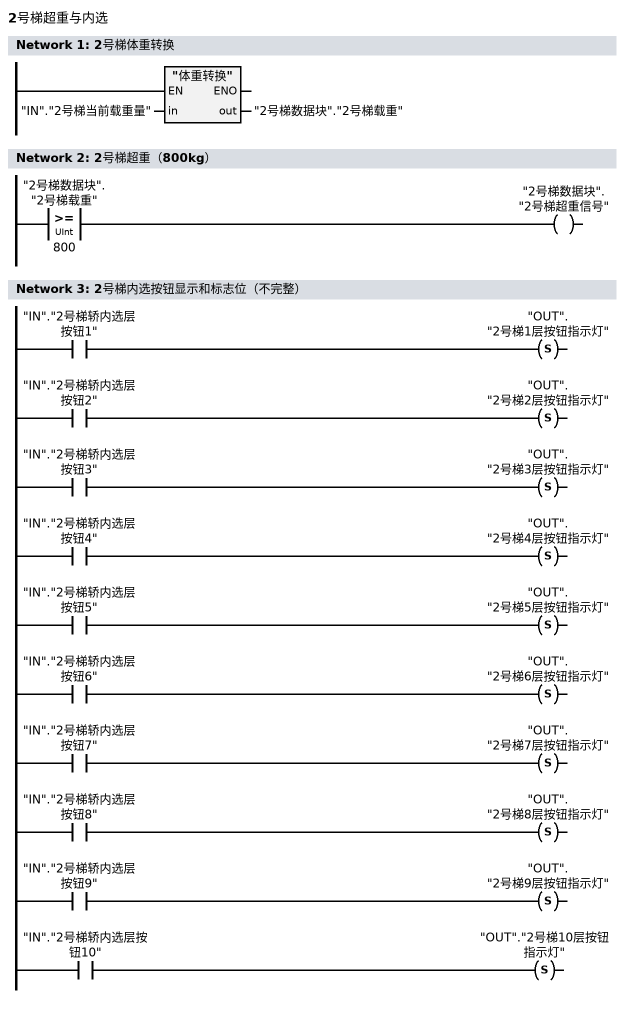
   RUNG wire#powerrail
      "体重转换"(in := "IN"."2号梯当前载重量", out => "2号梯数据块"."2号梯载重")
   END_RUNG
   // the same network as SCL:
   "体重转换"(in := "IN"."2号梯当前载重量", out => "2号梯数据块"."2号梯载重");
END_REGION

REGION Network 2: 2号梯超重（800kg）
   RUNG wire#powerrail
      { S7_Templates := "SrcType := UInt" } GE_Contact(in1 := "2号梯数据块"."2号梯载重", in2 := 800)
      Coil( "2号梯数据块"."2号梯超重信号" )
   END_RUNG
   // the same network as SCL:
   "2号梯数据块"."2号梯超重信号" := "2号梯数据块"."2号梯载重" >= 800;
END_REGION

REGION Network 3: 2号梯内选按钮显示和标志位（不完整）
   RUNG wire#powerrail
      Contact( "IN"."2号梯轿内选层按钮1" )
      S_Coil( "OUT"."2号梯1层按钮指示灯" )
   END_RUNG
   RUNG wire#powerrail
      Contact( "IN"."2号梯轿内选层按钮2" )
      S_Coil( "OUT"."2号梯2层按钮指示灯" )
   END_RUNG
   RUNG wire#powerrail
      Contact( "IN"."2号梯轿内选层按钮3" )
      S_Coil( "OUT"."2号梯3层按钮指示灯" )
   END_RUNG
   RUNG wire#powerrail
      Contact( "IN"."2号梯轿内选层按钮4" )
      S_Coil( "OUT"."2号梯4层按钮指示灯" )
   END_RUNG
   RUNG wire#powerrail
      Contact( "IN"."2号梯轿内选层按钮5" )
      S_Coil( "OUT"."2号梯5层按钮指示灯" )
   END_RUNG
   RUNG wire#powerrail
      Contact( "IN"."2号梯轿内选层按钮6" )
      S_Coil( "OUT"."2号梯6层按钮指示灯" )
   END_RUNG
   RUNG wire#powerrail
      Contact( "IN"."2号梯轿内选层按钮7" )
      S_Coil( "OUT"."2号梯7层按钮指示灯" )
   END_RUNG
   RUNG wire#powerrail
      Contact( "IN"."2号梯轿内选层按钮8" )
      S_Coil( "OUT"."2号梯8层按钮指示灯" )
   END_RUNG
   RUNG wire#powerrail
      Contact( "IN"."2号梯轿内选层按钮9" )
      S_Coil( "OUT"."2号梯9层按钮指示灯" )
   END_RUNG
   RUNG wire#powerrail
      Contact( "IN"."2号梯轿内选层按钮10" )
      S_Coil( "OUT"."2号梯10层按钮指示灯" )
   END_RUNG
   // the same network as SCL:
   IF "IN"."2号梯轿内选层按钮1" THEN "OUT"."2号梯1层按钮指示灯" := TRUE; END_IF;
   IF "IN"."2号梯轿内选层按钮2" THEN "OUT"."2号梯2层按钮指示灯" := TRUE; END_IF;
   IF "IN"."2号梯轿内选层按钮3" THEN "OUT"."2号梯3层按钮指示灯" := TRUE; END_IF;
   IF "IN"."2号梯轿内选层按钮4" THEN "OUT"."2号梯4层按钮指示灯" := TRUE; END_IF;
   IF "IN"."2号梯轿内选层按钮5" THEN "OUT"."2号梯5层按钮指示灯" := TRUE; END_IF;
   IF "IN"."2号梯轿内选层按钮6" THEN "OUT"."2号梯6层按钮指示灯" := TRUE; END_IF;
   IF "IN"."2号梯轿内选层按钮7" THEN "OUT"."2号梯7层按钮指示灯" := TRUE; END_IF;
   IF "IN"."2号梯轿内选层按钮8" THEN "OUT"."2号梯8层按钮指示灯" := TRUE; END_IF;
   IF "IN"."2号梯轿内选层按钮9" THEN "OUT"."2号梯9层按钮指示灯" := TRUE; END_IF;
   IF "IN"."2号梯轿内选层按钮10" THEN "OUT"."2号梯10层按钮指示灯" := TRUE; END_IF;
END_REGION
END_FUNCTION

FUNCTION "2号梯开关门控制" : Void   // FC27, LAD
{ S7_Optimized_Access := 'TRUE' }
VERSION : 0.1
BEGIN
END_FUNCTION

FUNCTION "2号梯楼层计数" : Void   // FC33, LAD
{ S7_Optimized_Access := 'TRUE' }
VERSION : 0.1
BEGIN
END_FUNCTION

FUNCTION "2号梯检修" : Void   // FC44, LAD
{ S7_Optimized_Access := 'TRUE' }
VERSION : 0.1
BEGIN
END_FUNCTION

FUNCTION "2号梯目标楼层与方向判断" : Void   // FC45, LAD
{ S7_Optimized_Access := 'TRUE' }
VERSION : 0.1
BEGIN
END_FUNCTION

FUNCTION "2号梯字节消除与记录" : Void   // FC46, LAD
{ S7_Optimized_Access := 'TRUE' }
VERSION : 0.1
BEGIN
END_FUNCTION

FUNCTION "2号梯启停控制" : Void   // FC59, LAD
{ S7_Optimized_Access := 'TRUE' }
VERSION : 0.1
BEGIN
END_FUNCTION

// folder: 3号梯

FUNCTION "3号梯初始化" : Void   // FC4, LAD
{ S7_Optimized_Access := 'TRUE' }
VERSION : 0.1
   VAR_INPUT
      初始化方向 : Bool;
      初始化楼层 : Byte;
   END_VAR
   VAR_TEMP   // added for the SCL form of the ladder/FBD networks
      _w1 : Bool;
      _w2 : Bool;
      _w3 : Bool;
      _w4 : Bool;
   END_VAR
BEGIN

REGION Network 1: 3号梯传参（方向+初始化楼层）
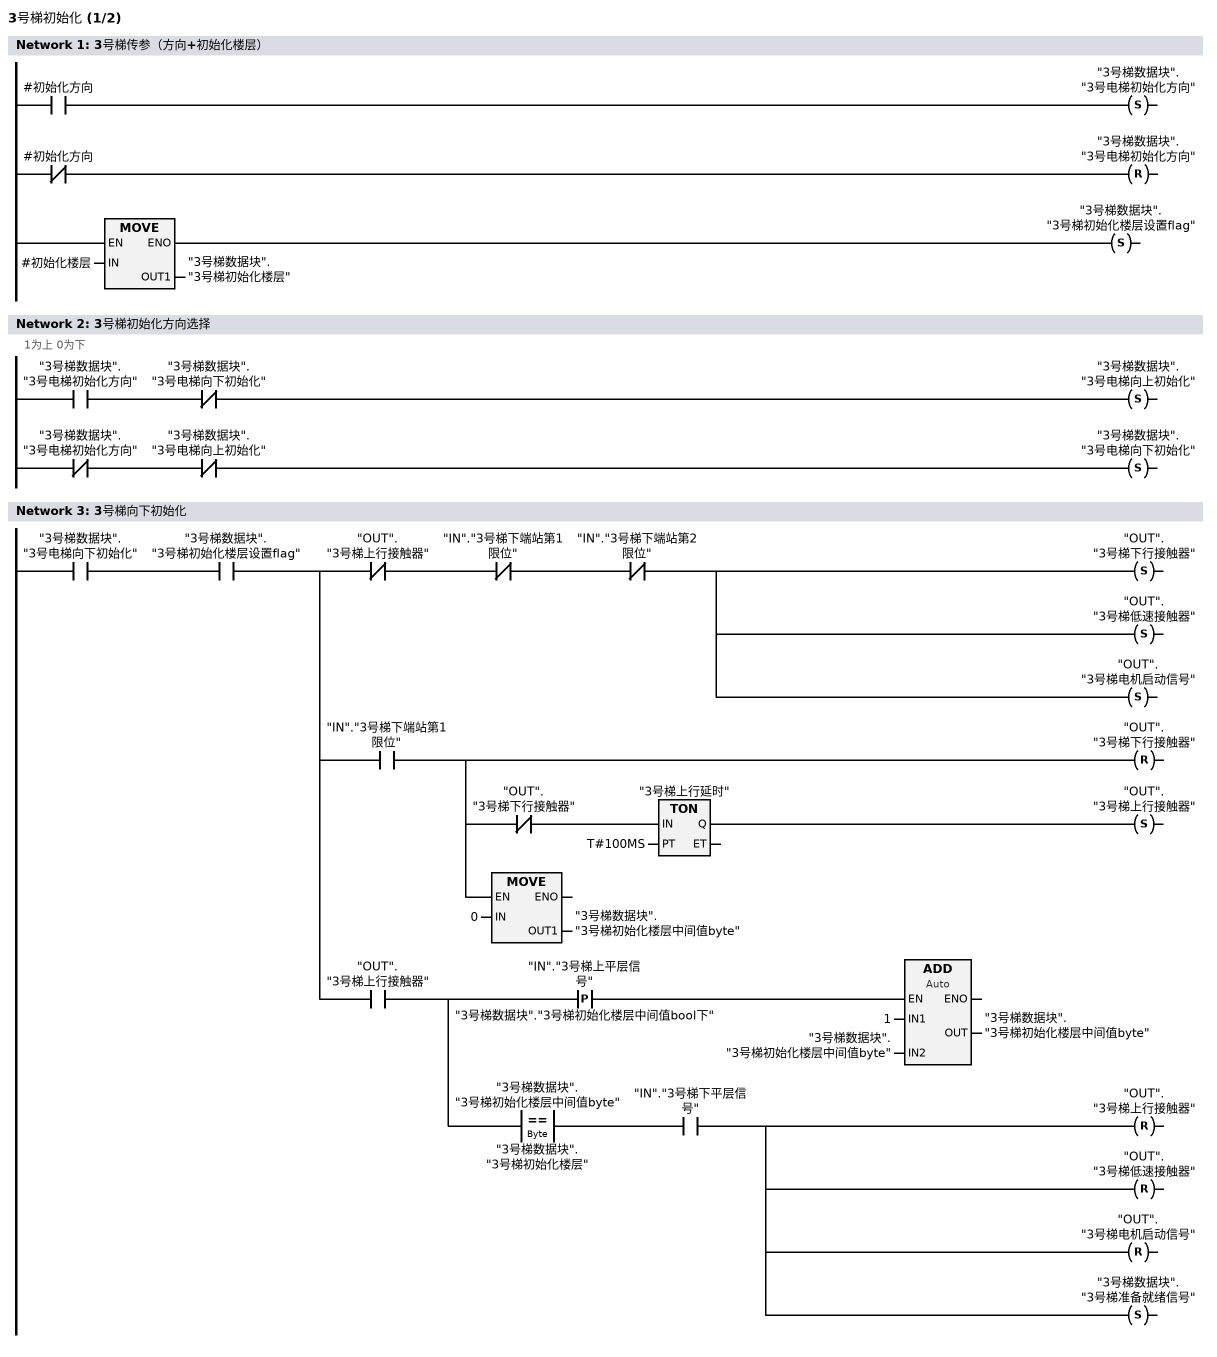
   RUNG wire#powerrail
      Contact( #初始化方向 )
      S_Coil( "3号梯数据块"."3号电梯初始化方向" )
   END_RUNG
   RUNG wire#powerrail
      I_Contact( #初始化方向 )
      R_Coil( "3号梯数据块"."3号电梯初始化方向" )
   END_RUNG
   RUNG wire#powerrail
      Move(in := #初始化楼层, out1 => "3号梯数据块"."3号梯初始化楼层")
      S_Coil( "3号梯数据块"."3号梯初始化楼层设置flag" )
   END_RUNG
   // the same network as SCL:
   IF #初始化方向 THEN "3号梯数据块"."3号电梯初始化方向" := TRUE; END_IF;
   IF NOT #初始化方向 THEN "3号梯数据块"."3号电梯初始化方向" := FALSE; END_IF;
   "3号梯数据块"."3号梯初始化楼层" := #初始化楼层;
   "3号梯数据块"."3号梯初始化楼层设置flag" := TRUE;
END_REGION

REGION Network 2: 3号梯初始化方向选择
   // 1为上 0为下
   RUNG wire#powerrail
      Contact( "3号梯数据块"."3号电梯初始化方向" )
      I_Contact( "3号梯数据块"."3号电梯向下初始化" )
      S_Coil( "3号梯数据块"."3号电梯向上初始化" )
   END_RUNG
   RUNG wire#powerrail
      I_Contact( "3号梯数据块"."3号电梯初始化方向" )
      I_Contact( "3号梯数据块"."3号电梯向上初始化" )
      S_Coil( "3号梯数据块"."3号电梯向下初始化" )
   END_RUNG
   // the same network as SCL:
   IF "3号梯数据块"."3号电梯初始化方向" AND NOT "3号梯数据块"."3号电梯向下初始化" THEN "3号梯数据块"."3号电梯向上初始化" := TRUE; END_IF;
   IF NOT "3号梯数据块"."3号电梯初始化方向" AND NOT "3号梯数据块"."3号电梯向上初始化" THEN "3号梯数据块"."3号电梯向下初始化" := TRUE; END_IF;
END_REGION

REGION Network 3: 3号梯向下初始化
   #_w1 := "3号梯数据块"."3号电梯向下初始化" AND "3号梯数据块"."3号梯初始化楼层设置flag";
   IF #_w1 AND NOT "OUT"."3号梯上行接触器" AND NOT "IN"."3号梯下端站第1限位" AND NOT "IN"."3号梯下端站第2限位" THEN
       "OUT"."3号梯下行接触器" := TRUE;
       "OUT"."3号梯低速接触器" := TRUE;
       "OUT"."3号梯电机启动信号" := TRUE;
   END_IF;
   #_w2 := #_w1 AND "IN"."3号梯下端站第1限位";
   IF #_w2 THEN "OUT"."3号梯下行接触器" := FALSE; END_IF;
   "3号梯上行延时".TON(IN := #_w2 AND NOT "OUT"."3号梯下行接触器", PT := T#100MS);
   IF "3号梯上行延时".Q THEN "OUT"."3号梯上行接触器" := TRUE; END_IF;
   IF #_w2 THEN "3号梯数据块"."3号梯初始化楼层中间值byte" := 0; END_IF;
   #_w3 := #_w1 AND "OUT"."3号梯上行接触器";
   #_w4 := #_w3 AND "IN"."3号梯上平层信号" AND NOT "3号梯数据块"."3号梯初始化楼层中间值bool下";   // rising edge of "IN"."3号梯上平层信号"
   "3号梯数据块"."3号梯初始化楼层中间值bool下" := "IN"."3号梯上平层信号";
   IF #_w4 THEN "3号梯数据块"."3号梯初始化楼层中间值byte" := 1 + "3号梯数据块"."3号梯初始化楼层中间值byte"; END_IF;
   IF #_w3 AND ("3号梯数据块"."3号梯初始化楼层中间值byte" = "3号梯数据块"."3号梯初始化楼层") AND "IN"."3号梯下平层信号" THEN
       "OUT"."3号梯上行接触器" := FALSE;
       "OUT"."3号梯低速接触器" := FALSE;
       "OUT"."3号梯电机启动信号" := FALSE;
       "3号梯数据块"."3号梯准备就绪信号" := TRUE;
   END_IF;
END_REGION

REGION Network 4: 3号梯向上初始化
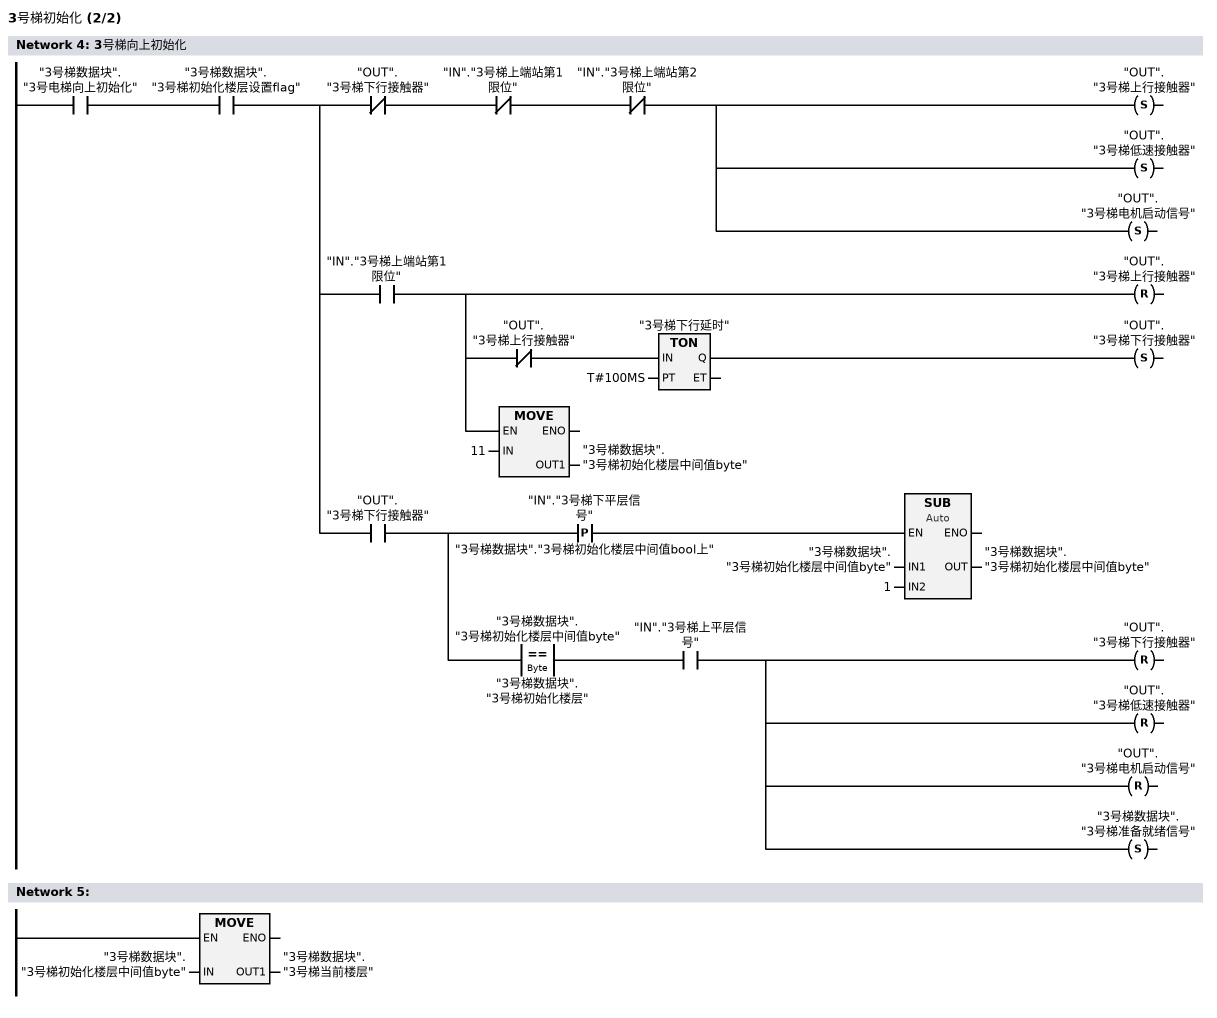
   #_w1 := "3号梯数据块"."3号电梯向上初始化" AND "3号梯数据块"."3号梯初始化楼层设置flag";
   IF #_w1 AND NOT "OUT"."3号梯下行接触器" AND NOT "IN"."3号梯上端站第1限位" AND NOT "IN"."3号梯上端站第2限位" THEN
       "OUT"."3号梯上行接触器" := TRUE;
       "OUT"."3号梯低速接触器" := TRUE;
       "OUT"."3号梯电机启动信号" := TRUE;
   END_IF;
   #_w2 := #_w1 AND "IN"."3号梯上端站第1限位";
   IF #_w2 THEN "OUT"."3号梯上行接触器" := FALSE; END_IF;
   "3号梯下行延时".TON(IN := #_w2 AND NOT "OUT"."3号梯上行接触器", PT := T#100MS);
   IF "3号梯下行延时".Q THEN "OUT"."3号梯下行接触器" := TRUE; END_IF;
   IF #_w2 THEN "3号梯数据块"."3号梯初始化楼层中间值byte" := 11; END_IF;
   #_w3 := #_w1 AND "OUT"."3号梯下行接触器";
   #_w4 := #_w3 AND "IN"."3号梯下平层信号" AND NOT "3号梯数据块"."3号梯初始化楼层中间值bool上";   // rising edge of "IN"."3号梯下平层信号"
   "3号梯数据块"."3号梯初始化楼层中间值bool上" := "IN"."3号梯下平层信号";
   IF #_w4 THEN "3号梯数据块"."3号梯初始化楼层中间值byte" := "3号梯数据块"."3号梯初始化楼层中间值byte" - 1; END_IF;
   IF #_w3 AND ("3号梯数据块"."3号梯初始化楼层中间值byte" = "3号梯数据块"."3号梯初始化楼层") AND "IN"."3号梯上平层信号" THEN
       "OUT"."3号梯下行接触器" := FALSE;
       "OUT"."3号梯低速接触器" := FALSE;
       "OUT"."3号梯电机启动信号" := FALSE;
       "3号梯数据块"."3号梯准备就绪信号" := TRUE;
   END_IF;
END_REGION

REGION Network 5
   RUNG wire#powerrail
      Move(in := "3号梯数据块"."3号梯初始化楼层中间值byte", out1 => "3号梯数据块"."3号梯当前楼层")
   END_RUNG
   // the same network as SCL:
   "3号梯数据块"."3号梯当前楼层" := "3号梯数据块"."3号梯初始化楼层中间值byte";
END_REGION
END_FUNCTION

FUNCTION "3号梯主函数" : Void   // FC10, LAD
{ S7_Optimized_Access := 'TRUE' }
VERSION : 0.1
BEGIN

REGION Network 1
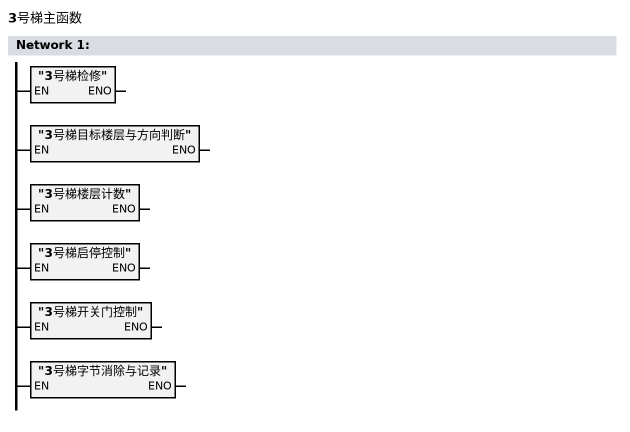
   RUNG wire#powerrail
      "3号梯检修"()
   END_RUNG
   RUNG wire#powerrail
      "3号梯目标楼层与方向判断"()
   END_RUNG
   RUNG wire#powerrail
      "3号梯楼层计数"()
   END_RUNG
   RUNG wire#powerrail
      "3号梯启停控制"()
   END_RUNG
   RUNG wire#powerrail
      "3号梯开关门控制"()
   END_RUNG
   RUNG wire#powerrail
      "3号梯字节消除与记录"()
   END_RUNG
   // the same network as SCL:
   "3号梯检修"();
   "3号梯目标楼层与方向判断"();
   "3号梯楼层计数"();
   "3号梯启停控制"();
   "3号梯开关门控制"();
   "3号梯字节消除与记录"();
END_REGION
END_FUNCTION

FUNCTION "3号梯运行监控模块" : Void   // FC16, LAD
{ S7_Optimized_Access := 'TRUE' }
VERSION : 0.1
BEGIN

REGION Network 1: 3号梯获取当前楼层设置标志位
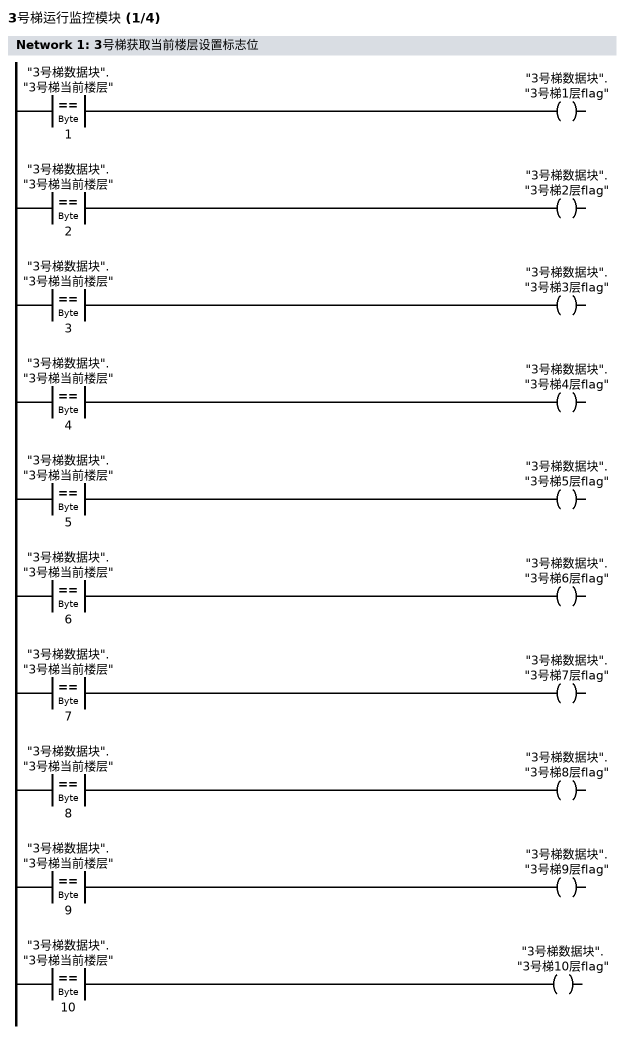
   RUNG wire#powerrail
      { S7_Templates := "SrcType := Byte" } EQ_Contact(in1 := "3号梯数据块"."3号梯当前楼层", in2 := 1)
      Coil( "3号梯数据块"."3号梯1层flag" )
   END_RUNG
   RUNG wire#powerrail
      { S7_Templates := "SrcType := Byte" } EQ_Contact(in1 := "3号梯数据块"."3号梯当前楼层", in2 := 2)
      Coil( "3号梯数据块"."3号梯2层flag" )
   END_RUNG
   RUNG wire#powerrail
      { S7_Templates := "SrcType := Byte" } EQ_Contact(in1 := "3号梯数据块"."3号梯当前楼层", in2 := 3)
      Coil( "3号梯数据块"."3号梯3层flag" )
   END_RUNG
   RUNG wire#powerrail
      { S7_Templates := "SrcType := Byte" } EQ_Contact(in1 := "3号梯数据块"."3号梯当前楼层", in2 := 4)
      Coil( "3号梯数据块"."3号梯4层flag" )
   END_RUNG
   RUNG wire#powerrail
      { S7_Templates := "SrcType := Byte" } EQ_Contact(in1 := "3号梯数据块"."3号梯当前楼层", in2 := 5)
      Coil( "3号梯数据块"."3号梯5层flag" )
   END_RUNG
   RUNG wire#powerrail
      { S7_Templates := "SrcType := Byte" } EQ_Contact(in1 := "3号梯数据块"."3号梯当前楼层", in2 := 6)
      Coil( "3号梯数据块"."3号梯6层flag" )
   END_RUNG
   RUNG wire#powerrail
      { S7_Templates := "SrcType := Byte" } EQ_Contact(in1 := "3号梯数据块"."3号梯当前楼层", in2 := 7)
      Coil( "3号梯数据块"."3号梯7层flag" )
   END_RUNG
   RUNG wire#powerrail
      { S7_Templates := "SrcType := Byte" } EQ_Contact(in1 := "3号梯数据块"."3号梯当前楼层", in2 := 8)
      Coil( "3号梯数据块"."3号梯8层flag" )
   END_RUNG
   RUNG wire#powerrail
      { S7_Templates := "SrcType := Byte" } EQ_Contact(in1 := "3号梯数据块"."3号梯当前楼层", in2 := 9)
      Coil( "3号梯数据块"."3号梯9层flag" )
   END_RUNG
   RUNG wire#powerrail
      { S7_Templates := "SrcType := Byte" } EQ_Contact(in1 := "3号梯数据块"."3号梯当前楼层", in2 := 10)
      Coil( "3号梯数据块"."3号梯10层flag" )
   END_RUNG
   // the same network as SCL:
   "3号梯数据块"."3号梯1层flag" := "3号梯数据块"."3号梯当前楼层" = 1;
   "3号梯数据块"."3号梯2层flag" := "3号梯数据块"."3号梯当前楼层" = 2;
   "3号梯数据块"."3号梯3层flag" := "3号梯数据块"."3号梯当前楼层" = 3;
   "3号梯数据块"."3号梯4层flag" := "3号梯数据块"."3号梯当前楼层" = 4;
   "3号梯数据块"."3号梯5层flag" := "3号梯数据块"."3号梯当前楼层" = 5;
   "3号梯数据块"."3号梯6层flag" := "3号梯数据块"."3号梯当前楼层" = 6;
   "3号梯数据块"."3号梯7层flag" := "3号梯数据块"."3号梯当前楼层" = 7;
   "3号梯数据块"."3号梯8层flag" := "3号梯数据块"."3号梯当前楼层" = 8;
   "3号梯数据块"."3号梯9层flag" := "3号梯数据块"."3号梯当前楼层" = 9;
   "3号梯数据块"."3号梯10层flag" := "3号梯数据块"."3号梯当前楼层" = 10;
END_REGION

REGION Network 2: 3号梯楼层led_a显示
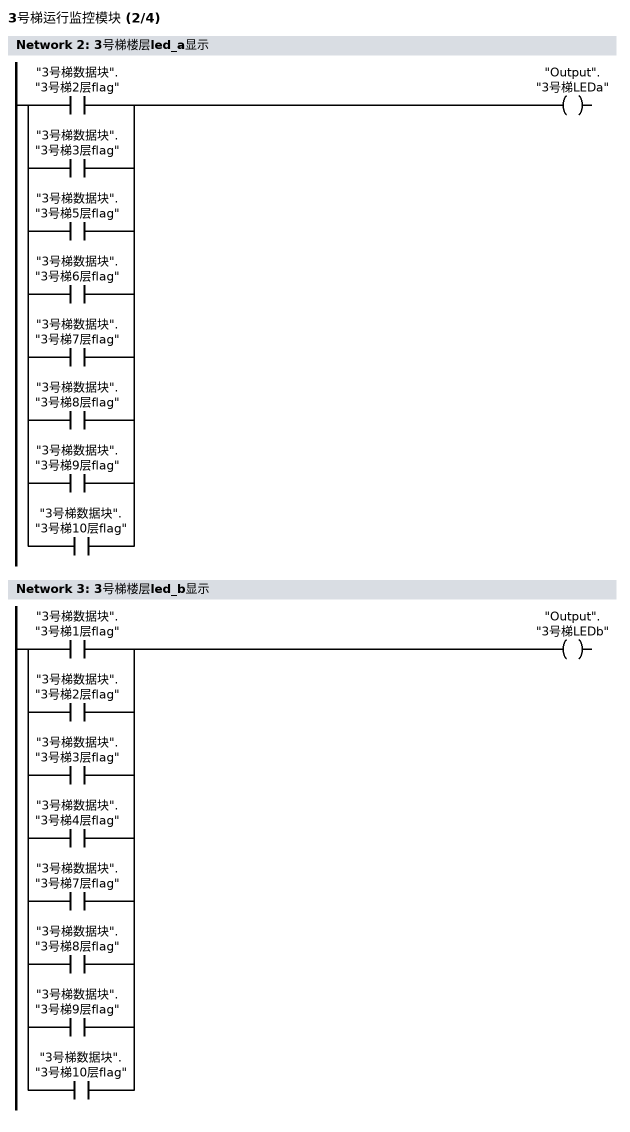
   RUNG wire#powerrail
      Contact( "3号梯数据块"."3号梯2层flag" )
      wire#w1
      Coil( "Output"."3号梯LEDa" )
   END_RUNG
   RUNG wire#powerrail
      Contact( "3号梯数据块"."3号梯3层flag" )
   END_RUNG wire#w1
   RUNG wire#powerrail
      Contact( "3号梯数据块"."3号梯5层flag" )
   END_RUNG wire#w1
   RUNG wire#powerrail
      Contact( "3号梯数据块"."3号梯6层flag" )
   END_RUNG wire#w1
   RUNG wire#powerrail
      Contact( "3号梯数据块"."3号梯7层flag" )
   END_RUNG wire#w1
   RUNG wire#powerrail
      Contact( "3号梯数据块"."3号梯8层flag" )
   END_RUNG wire#w1
   RUNG wire#powerrail
      Contact( "3号梯数据块"."3号梯9层flag" )
   END_RUNG wire#w1
   RUNG wire#powerrail
      Contact( "3号梯数据块"."3号梯10层flag" )
   END_RUNG wire#w1
   // the same network as SCL:
   "Output"."3号梯LEDa" := "3号梯数据块"."3号梯2层flag" OR "3号梯数据块"."3号梯3层flag" OR "3号梯数据块"."3号梯5层flag" OR "3号梯数据块"."3号梯6层flag" OR "3号梯数据块"."3号梯7层flag" OR "3号梯数据块"."3号梯8层flag" OR "3号梯数据块"."3号梯9层flag" OR "3号梯数据块"."3号梯10层flag";
END_REGION

REGION Network 3: 3号梯楼层led_b显示
   RUNG wire#powerrail
      Contact( "3号梯数据块"."3号梯1层flag" )
      wire#w1
      Coil( "Output"."3号梯LEDb" )
   END_RUNG
   RUNG wire#powerrail
      Contact( "3号梯数据块"."3号梯2层flag" )
   END_RUNG wire#w1
   RUNG wire#powerrail
      Contact( "3号梯数据块"."3号梯3层flag" )
   END_RUNG wire#w1
   RUNG wire#powerrail
      Contact( "3号梯数据块"."3号梯4层flag" )
   END_RUNG wire#w1
   RUNG wire#powerrail
      Contact( "3号梯数据块"."3号梯7层flag" )
   END_RUNG wire#w1
   RUNG wire#powerrail
      Contact( "3号梯数据块"."3号梯8层flag" )
   END_RUNG wire#w1
   RUNG wire#powerrail
      Contact( "3号梯数据块"."3号梯9层flag" )
   END_RUNG wire#w1
   RUNG wire#powerrail
      Contact( "3号梯数据块"."3号梯10层flag" )
   END_RUNG wire#w1
   // the same network as SCL:
   "Output"."3号梯LEDb" := "3号梯数据块"."3号梯1层flag" OR "3号梯数据块"."3号梯2层flag" OR "3号梯数据块"."3号梯3层flag" OR "3号梯数据块"."3号梯4层flag" OR "3号梯数据块"."3号梯7层flag" OR "3号梯数据块"."3号梯8层flag" OR "3号梯数据块"."3号梯9层flag" OR "3号梯数据块"."3号梯10层flag";
END_REGION

REGION Network 4: 3号梯楼层led_c显示
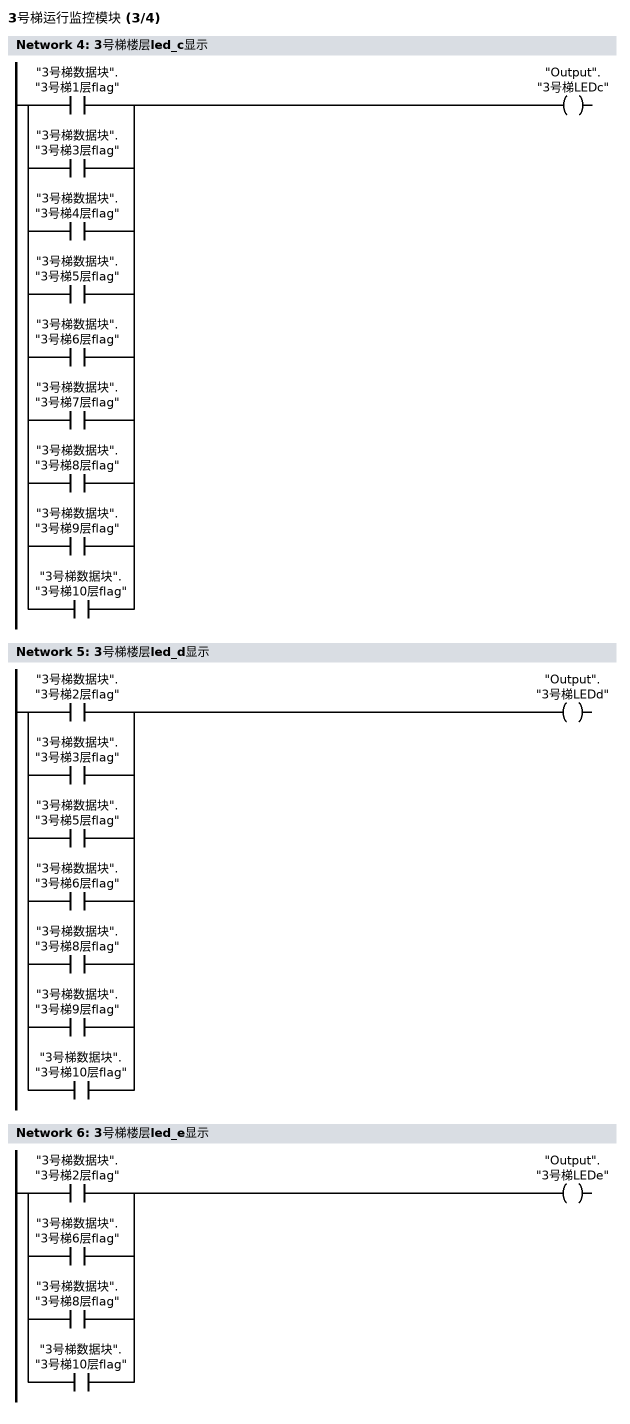
   RUNG wire#powerrail
      Contact( "3号梯数据块"."3号梯1层flag" )
      wire#w1
      Coil( "Output"."3号梯LEDc" )
   END_RUNG
   RUNG wire#powerrail
      Contact( "3号梯数据块"."3号梯3层flag" )
   END_RUNG wire#w1
   RUNG wire#powerrail
      Contact( "3号梯数据块"."3号梯4层flag" )
   END_RUNG wire#w1
   RUNG wire#powerrail
      Contact( "3号梯数据块"."3号梯5层flag" )
   END_RUNG wire#w1
   RUNG wire#powerrail
      Contact( "3号梯数据块"."3号梯6层flag" )
   END_RUNG wire#w1
   RUNG wire#powerrail
      Contact( "3号梯数据块"."3号梯7层flag" )
   END_RUNG wire#w1
   RUNG wire#powerrail
      Contact( "3号梯数据块"."3号梯8层flag" )
   END_RUNG wire#w1
   RUNG wire#powerrail
      Contact( "3号梯数据块"."3号梯9层flag" )
   END_RUNG wire#w1
   RUNG wire#powerrail
      Contact( "3号梯数据块"."3号梯10层flag" )
   END_RUNG wire#w1
   // the same network as SCL:
   "Output"."3号梯LEDc" := "3号梯数据块"."3号梯1层flag" OR "3号梯数据块"."3号梯3层flag" OR "3号梯数据块"."3号梯4层flag" OR "3号梯数据块"."3号梯5层flag" OR "3号梯数据块"."3号梯6层flag" OR "3号梯数据块"."3号梯7层flag" OR "3号梯数据块"."3号梯8层flag" OR "3号梯数据块"."3号梯9层flag" OR "3号梯数据块"."3号梯10层flag";
END_REGION

REGION Network 5: 3号梯楼层led_d显示
   RUNG wire#powerrail
      Contact( "3号梯数据块"."3号梯2层flag" )
      wire#w1
      Coil( "Output"."3号梯LEDd" )
   END_RUNG
   RUNG wire#powerrail
      Contact( "3号梯数据块"."3号梯3层flag" )
   END_RUNG wire#w1
   RUNG wire#powerrail
      Contact( "3号梯数据块"."3号梯5层flag" )
   END_RUNG wire#w1
   RUNG wire#powerrail
      Contact( "3号梯数据块"."3号梯6层flag" )
   END_RUNG wire#w1
   RUNG wire#powerrail
      Contact( "3号梯数据块"."3号梯8层flag" )
   END_RUNG wire#w1
   RUNG wire#powerrail
      Contact( "3号梯数据块"."3号梯9层flag" )
   END_RUNG wire#w1
   RUNG wire#powerrail
      Contact( "3号梯数据块"."3号梯10层flag" )
   END_RUNG wire#w1
   // the same network as SCL:
   "Output"."3号梯LEDd" := "3号梯数据块"."3号梯2层flag" OR "3号梯数据块"."3号梯3层flag" OR "3号梯数据块"."3号梯5层flag" OR "3号梯数据块"."3号梯6层flag" OR "3号梯数据块"."3号梯8层flag" OR "3号梯数据块"."3号梯9层flag" OR "3号梯数据块"."3号梯10层flag";
END_REGION

REGION Network 6: 3号梯楼层led_e显示
   RUNG wire#powerrail
      Contact( "3号梯数据块"."3号梯2层flag" )
      wire#w1
      Coil( "Output"."3号梯LEDe" )
   END_RUNG
   RUNG wire#powerrail
      Contact( "3号梯数据块"."3号梯6层flag" )
   END_RUNG wire#w1
   RUNG wire#powerrail
      Contact( "3号梯数据块"."3号梯8层flag" )
   END_RUNG wire#w1
   RUNG wire#powerrail
      Contact( "3号梯数据块"."3号梯10层flag" )
   END_RUNG wire#w1
   // the same network as SCL:
   "Output"."3号梯LEDe" := "3号梯数据块"."3号梯2层flag" OR "3号梯数据块"."3号梯6层flag" OR "3号梯数据块"."3号梯8层flag" OR "3号梯数据块"."3号梯10层flag";
END_REGION

REGION Network 7: 3号梯楼层led_f显示
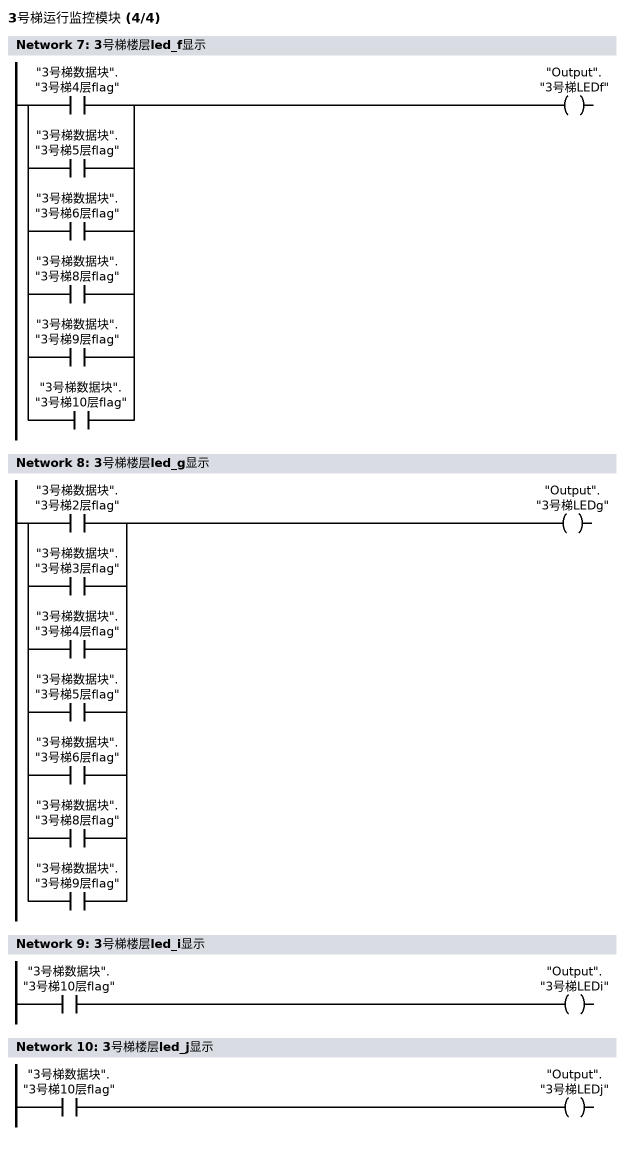
   RUNG wire#powerrail
      Contact( "3号梯数据块"."3号梯4层flag" )
      wire#w1
      Coil( "Output"."3号梯LEDf" )
   END_RUNG
   RUNG wire#powerrail
      Contact( "3号梯数据块"."3号梯5层flag" )
   END_RUNG wire#w1
   RUNG wire#powerrail
      Contact( "3号梯数据块"."3号梯6层flag" )
   END_RUNG wire#w1
   RUNG wire#powerrail
      Contact( "3号梯数据块"."3号梯8层flag" )
   END_RUNG wire#w1
   RUNG wire#powerrail
      Contact( "3号梯数据块"."3号梯9层flag" )
   END_RUNG wire#w1
   RUNG wire#powerrail
      Contact( "3号梯数据块"."3号梯10层flag" )
   END_RUNG wire#w1
   // the same network as SCL:
   "Output"."3号梯LEDf" := "3号梯数据块"."3号梯4层flag" OR "3号梯数据块"."3号梯5层flag" OR "3号梯数据块"."3号梯6层flag" OR "3号梯数据块"."3号梯8层flag" OR "3号梯数据块"."3号梯9层flag" OR "3号梯数据块"."3号梯10层flag";
END_REGION

REGION Network 8: 3号梯楼层led_g显示
   RUNG wire#powerrail
      Contact( "3号梯数据块"."3号梯2层flag" )
      wire#w1
      Coil( "Output"."3号梯LEDg" )
   END_RUNG
   RUNG wire#powerrail
      Contact( "3号梯数据块"."3号梯3层flag" )
   END_RUNG wire#w1
   RUNG wire#powerrail
      Contact( "3号梯数据块"."3号梯4层flag" )
   END_RUNG wire#w1
   RUNG wire#powerrail
      Contact( "3号梯数据块"."3号梯5层flag" )
   END_RUNG wire#w1
   RUNG wire#powerrail
      Contact( "3号梯数据块"."3号梯6层flag" )
   END_RUNG wire#w1
   RUNG wire#powerrail
      Contact( "3号梯数据块"."3号梯8层flag" )
   END_RUNG wire#w1
   RUNG wire#powerrail
      Contact( "3号梯数据块"."3号梯9层flag" )
   END_RUNG wire#w1
   // the same network as SCL:
   "Output"."3号梯LEDg" := "3号梯数据块"."3号梯2层flag" OR "3号梯数据块"."3号梯3层flag" OR "3号梯数据块"."3号梯4层flag" OR "3号梯数据块"."3号梯5层flag" OR "3号梯数据块"."3号梯6层flag" OR "3号梯数据块"."3号梯8层flag" OR "3号梯数据块"."3号梯9层flag";
END_REGION

REGION Network 9: 3号梯楼层led_i显示
   RUNG wire#powerrail
      Contact( "3号梯数据块"."3号梯10层flag" )
      Coil( "Output"."3号梯LEDi" )
   END_RUNG
   // the same network as SCL:
   "Output"."3号梯LEDi" := "3号梯数据块"."3号梯10层flag";
END_REGION

REGION Network 10: 3号梯楼层led_j显示
   RUNG wire#powerrail
      Contact( "3号梯数据块"."3号梯10层flag" )
      Coil( "Output"."3号梯LEDj" )
   END_RUNG
   // the same network as SCL:
   "Output"."3号梯LEDj" := "3号梯数据块"."3号梯10层flag";
END_REGION
END_FUNCTION

FUNCTION "3号梯开关门控制" : Void   // FC28, LAD
{ S7_Optimized_Access := 'TRUE' }
VERSION : 0.1
BEGIN
END_FUNCTION

FUNCTION "3号梯楼层计数" : Void   // FC34, LAD
{ S7_Optimized_Access := 'TRUE' }
VERSION : 0.1
BEGIN
END_FUNCTION

FUNCTION "3号梯超重与内选" : Void   // FC47, LAD
{ S7_Optimized_Access := 'TRUE' }
VERSION : 0.1
BEGIN
END_FUNCTION

FUNCTION "3号梯检修" : Void   // FC48, LAD
{ S7_Optimized_Access := 'TRUE' }
VERSION : 0.1
BEGIN
END_FUNCTION

FUNCTION "3号梯目标楼层与方向判断" : Void   // FC49, LAD
{ S7_Optimized_Access := 'TRUE' }
VERSION : 0.1
BEGIN
END_FUNCTION

FUNCTION "3号梯字节消除与记录" : Void   // FC50, LAD
{ S7_Optimized_Access := 'TRUE' }
VERSION : 0.1
BEGIN
END_FUNCTION

FUNCTION "3号梯启停控制" : Void   // FC60, LAD
{ S7_Optimized_Access := 'TRUE' }
VERSION : 0.1
BEGIN
END_FUNCTION

// folder: 4号梯

FUNCTION "4号梯初始化" : Void   // FC5, LAD
{ S7_Optimized_Access := 'TRUE' }
VERSION : 0.1
   VAR_INPUT
      初始化方向 : Bool;
      初始化楼层 : Byte;
   END_VAR
   VAR_TEMP   // added for the SCL form of the ladder/FBD networks
      _w1 : Bool;
      _w2 : Bool;
      _w3 : Bool;
      _w4 : Bool;
   END_VAR
BEGIN

REGION Network 1: 4号梯传参（方向+初始化楼层）
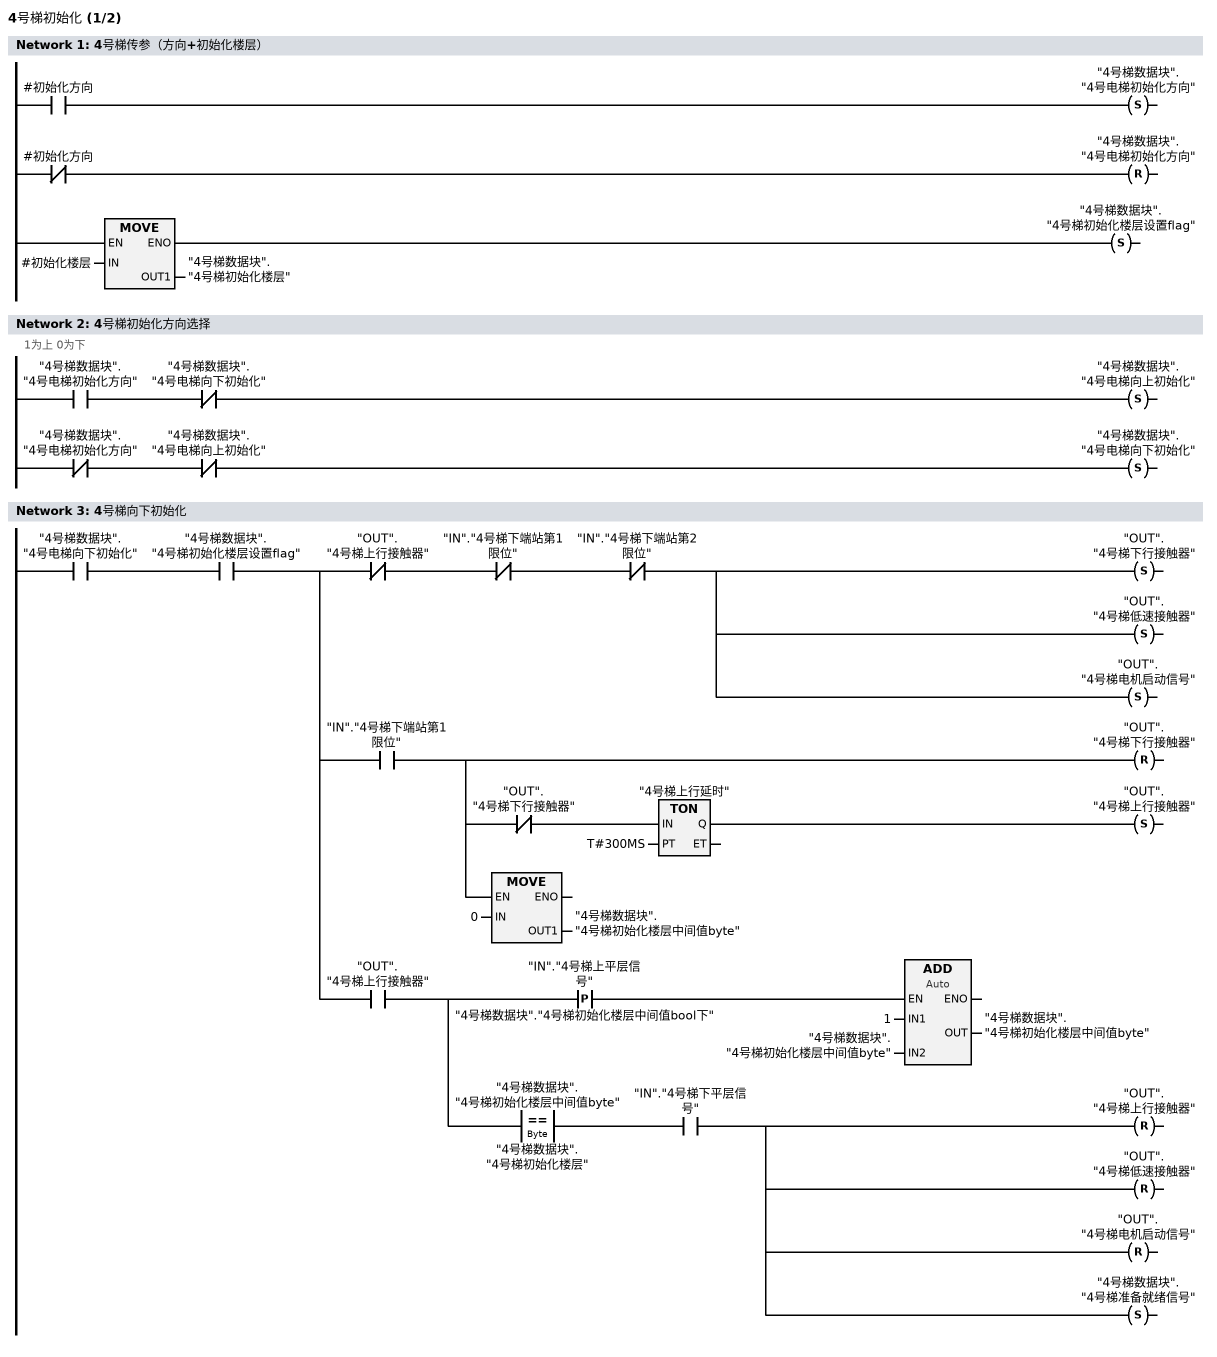
   RUNG wire#powerrail
      Contact( #初始化方向 )
      S_Coil( "4号梯数据块"."4号电梯初始化方向" )
   END_RUNG
   RUNG wire#powerrail
      I_Contact( #初始化方向 )
      R_Coil( "4号梯数据块"."4号电梯初始化方向" )
   END_RUNG
   RUNG wire#powerrail
      Move(in := #初始化楼层, out1 => "4号梯数据块"."4号梯初始化楼层")
      S_Coil( "4号梯数据块"."4号梯初始化楼层设置flag" )
   END_RUNG
   // the same network as SCL:
   IF #初始化方向 THEN "4号梯数据块"."4号电梯初始化方向" := TRUE; END_IF;
   IF NOT #初始化方向 THEN "4号梯数据块"."4号电梯初始化方向" := FALSE; END_IF;
   "4号梯数据块"."4号梯初始化楼层" := #初始化楼层;
   "4号梯数据块"."4号梯初始化楼层设置flag" := TRUE;
END_REGION

REGION Network 2: 4号梯初始化方向选择
   // 1为上 0为下
   RUNG wire#powerrail
      Contact( "4号梯数据块"."4号电梯初始化方向" )
      I_Contact( "4号梯数据块"."4号电梯向下初始化" )
      S_Coil( "4号梯数据块"."4号电梯向上初始化" )
   END_RUNG
   RUNG wire#powerrail
      I_Contact( "4号梯数据块"."4号电梯初始化方向" )
      I_Contact( "4号梯数据块"."4号电梯向上初始化" )
      S_Coil( "4号梯数据块"."4号电梯向下初始化" )
   END_RUNG
   // the same network as SCL:
   IF "4号梯数据块"."4号电梯初始化方向" AND NOT "4号梯数据块"."4号电梯向下初始化" THEN "4号梯数据块"."4号电梯向上初始化" := TRUE; END_IF;
   IF NOT "4号梯数据块"."4号电梯初始化方向" AND NOT "4号梯数据块"."4号电梯向上初始化" THEN "4号梯数据块"."4号电梯向下初始化" := TRUE; END_IF;
END_REGION

REGION Network 3: 4号梯向下初始化
   #_w1 := "4号梯数据块"."4号电梯向下初始化" AND "4号梯数据块"."4号梯初始化楼层设置flag";
   IF #_w1 AND NOT "OUT"."4号梯上行接触器" AND NOT "IN"."4号梯下端站第1限位" AND NOT "IN"."4号梯下端站第2限位" THEN
       "OUT"."4号梯下行接触器" := TRUE;
       "OUT"."4号梯低速接触器" := TRUE;
       "OUT"."4号梯电机启动信号" := TRUE;
   END_IF;
   #_w2 := #_w1 AND "IN"."4号梯下端站第1限位";
   IF #_w2 THEN "OUT"."4号梯下行接触器" := FALSE; END_IF;
   "4号梯上行延时".TON(IN := #_w2 AND NOT "OUT"."4号梯下行接触器", PT := T#300MS);
   IF "4号梯上行延时".Q THEN "OUT"."4号梯上行接触器" := TRUE; END_IF;
   IF #_w2 THEN "4号梯数据块"."4号梯初始化楼层中间值byte" := 0; END_IF;
   #_w3 := #_w1 AND "OUT"."4号梯上行接触器";
   #_w4 := #_w3 AND "IN"."4号梯上平层信号" AND NOT "4号梯数据块"."4号梯初始化楼层中间值bool下";   // rising edge of "IN"."4号梯上平层信号"
   "4号梯数据块"."4号梯初始化楼层中间值bool下" := "IN"."4号梯上平层信号";
   IF #_w4 THEN "4号梯数据块"."4号梯初始化楼层中间值byte" := 1 + "4号梯数据块"."4号梯初始化楼层中间值byte"; END_IF;
   IF #_w3 AND ("4号梯数据块"."4号梯初始化楼层中间值byte" = "4号梯数据块"."4号梯初始化楼层") AND "IN"."4号梯下平层信号" THEN
       "OUT"."4号梯上行接触器" := FALSE;
       "OUT"."4号梯低速接触器" := FALSE;
       "OUT"."4号梯电机启动信号" := FALSE;
       "4号梯数据块"."4号梯准备就绪信号" := TRUE;
   END_IF;
END_REGION

REGION Network 4: 4号梯向上初始化
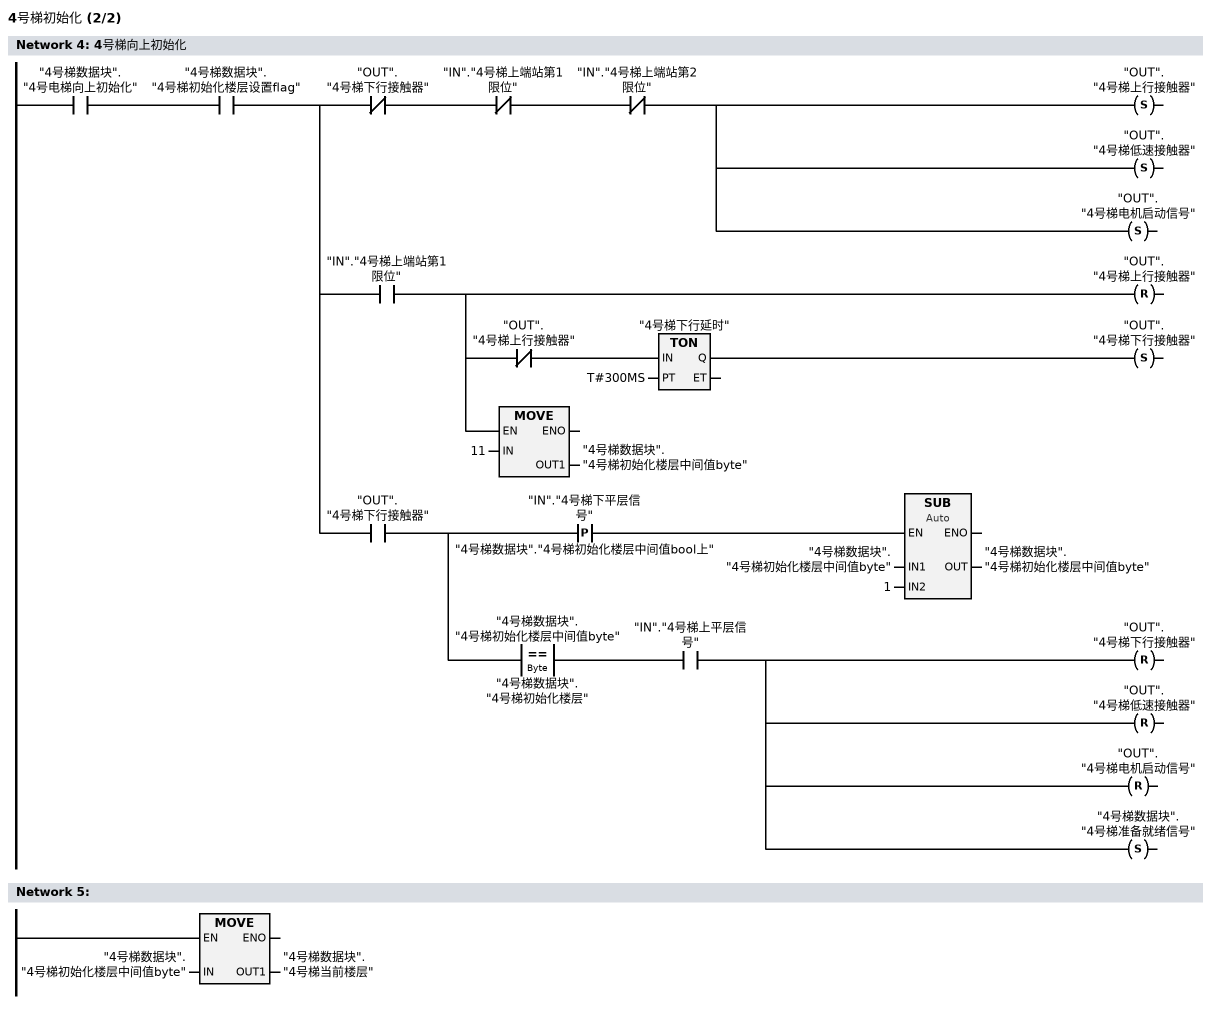
   #_w1 := "4号梯数据块"."4号电梯向上初始化" AND "4号梯数据块"."4号梯初始化楼层设置flag";
   IF #_w1 AND NOT "OUT"."4号梯下行接触器" AND NOT "IN"."4号梯上端站第1限位" AND NOT "IN"."4号梯上端站第2限位" THEN
       "OUT"."4号梯上行接触器" := TRUE;
       "OUT"."4号梯低速接触器" := TRUE;
       "OUT"."4号梯电机启动信号" := TRUE;
   END_IF;
   #_w2 := #_w1 AND "IN"."4号梯上端站第1限位";
   IF #_w2 THEN "OUT"."4号梯上行接触器" := FALSE; END_IF;
   "4号梯下行延时".TON(IN := #_w2 AND NOT "OUT"."4号梯上行接触器", PT := T#300MS);
   IF "4号梯下行延时".Q THEN "OUT"."4号梯下行接触器" := TRUE; END_IF;
   IF #_w2 THEN "4号梯数据块"."4号梯初始化楼层中间值byte" := 11; END_IF;
   #_w3 := #_w1 AND "OUT"."4号梯下行接触器";
   #_w4 := #_w3 AND "IN"."4号梯下平层信号" AND NOT "4号梯数据块"."4号梯初始化楼层中间值bool上";   // rising edge of "IN"."4号梯下平层信号"
   "4号梯数据块"."4号梯初始化楼层中间值bool上" := "IN"."4号梯下平层信号";
   IF #_w4 THEN "4号梯数据块"."4号梯初始化楼层中间值byte" := "4号梯数据块"."4号梯初始化楼层中间值byte" - 1; END_IF;
   IF #_w3 AND ("4号梯数据块"."4号梯初始化楼层中间值byte" = "4号梯数据块"."4号梯初始化楼层") AND "IN"."4号梯上平层信号" THEN
       "OUT"."4号梯下行接触器" := FALSE;
       "OUT"."4号梯低速接触器" := FALSE;
       "OUT"."4号梯电机启动信号" := FALSE;
       "4号梯数据块"."4号梯准备就绪信号" := TRUE;
   END_IF;
END_REGION

REGION Network 5
   RUNG wire#powerrail
      Move(in := "4号梯数据块"."4号梯初始化楼层中间值byte", out1 => "4号梯数据块"."4号梯当前楼层")
   END_RUNG
   // the same network as SCL:
   "4号梯数据块"."4号梯当前楼层" := "4号梯数据块"."4号梯初始化楼层中间值byte";
END_REGION
END_FUNCTION

FUNCTION "4号梯主函数" : Void   // FC11, LAD
{ S7_Optimized_Access := 'TRUE' }
VERSION : 0.1
BEGIN

REGION Network 1
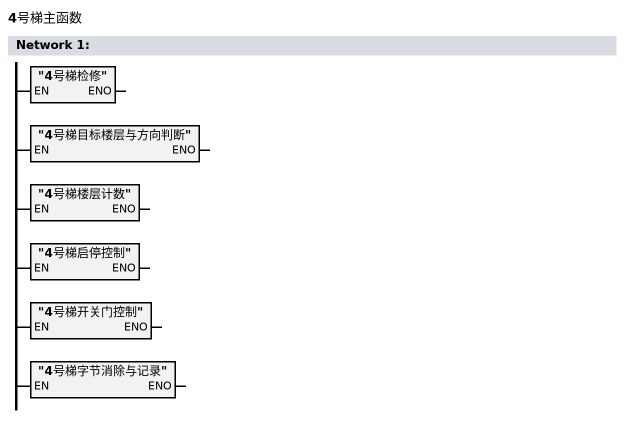
   RUNG wire#powerrail
      "4号梯检修"()
   END_RUNG
   RUNG wire#powerrail
      "4号梯目标楼层与方向判断"()
   END_RUNG
   RUNG wire#powerrail
      "4号梯楼层计数"()
   END_RUNG
   RUNG wire#powerrail
      "4号梯启停控制"()
   END_RUNG
   RUNG wire#powerrail
      "4号梯开关门控制"()
   END_RUNG
   RUNG wire#powerrail
      "4号梯字节消除与记录"()
   END_RUNG
   // the same network as SCL:
   "4号梯检修"();
   "4号梯目标楼层与方向判断"();
   "4号梯楼层计数"();
   "4号梯启停控制"();
   "4号梯开关门控制"();
   "4号梯字节消除与记录"();
END_REGION
END_FUNCTION

FUNCTION "4号梯运行监控模块" : Void   // FC17, LAD
{ S7_Optimized_Access := 'TRUE' }
VERSION : 0.1
BEGIN

REGION Network 1: 4号梯获取当前楼层设置标志位
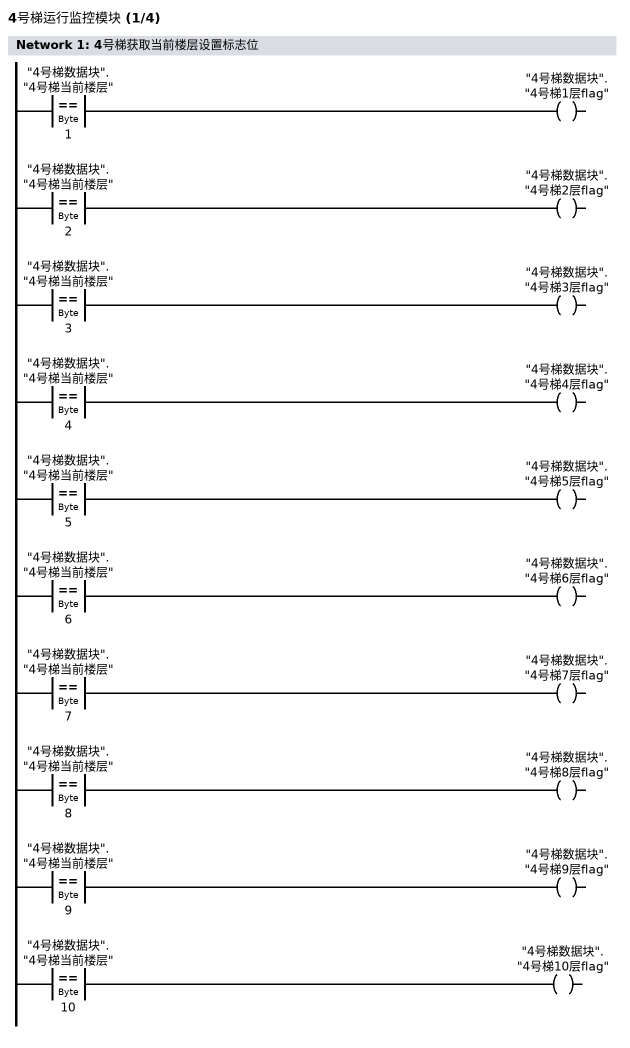
   RUNG wire#powerrail
      { S7_Templates := "SrcType := Byte" } EQ_Contact(in1 := "4号梯数据块"."4号梯当前楼层", in2 := 1)
      Coil( "4号梯数据块"."4号梯1层flag" )
   END_RUNG
   RUNG wire#powerrail
      { S7_Templates := "SrcType := Byte" } EQ_Contact(in1 := "4号梯数据块"."4号梯当前楼层", in2 := 2)
      Coil( "4号梯数据块"."4号梯2层flag" )
   END_RUNG
   RUNG wire#powerrail
      { S7_Templates := "SrcType := Byte" } EQ_Contact(in1 := "4号梯数据块"."4号梯当前楼层", in2 := 3)
      Coil( "4号梯数据块"."4号梯3层flag" )
   END_RUNG
   RUNG wire#powerrail
      { S7_Templates := "SrcType := Byte" } EQ_Contact(in1 := "4号梯数据块"."4号梯当前楼层", in2 := 4)
      Coil( "4号梯数据块"."4号梯4层flag" )
   END_RUNG
   RUNG wire#powerrail
      { S7_Templates := "SrcType := Byte" } EQ_Contact(in1 := "4号梯数据块"."4号梯当前楼层", in2 := 5)
      Coil( "4号梯数据块"."4号梯5层flag" )
   END_RUNG
   RUNG wire#powerrail
      { S7_Templates := "SrcType := Byte" } EQ_Contact(in1 := "4号梯数据块"."4号梯当前楼层", in2 := 6)
      Coil( "4号梯数据块"."4号梯6层flag" )
   END_RUNG
   RUNG wire#powerrail
      { S7_Templates := "SrcType := Byte" } EQ_Contact(in1 := "4号梯数据块"."4号梯当前楼层", in2 := 7)
      Coil( "4号梯数据块"."4号梯7层flag" )
   END_RUNG
   RUNG wire#powerrail
      { S7_Templates := "SrcType := Byte" } EQ_Contact(in1 := "4号梯数据块"."4号梯当前楼层", in2 := 8)
      Coil( "4号梯数据块"."4号梯8层flag" )
   END_RUNG
   RUNG wire#powerrail
      { S7_Templates := "SrcType := Byte" } EQ_Contact(in1 := "4号梯数据块"."4号梯当前楼层", in2 := 9)
      Coil( "4号梯数据块"."4号梯9层flag" )
   END_RUNG
   RUNG wire#powerrail
      { S7_Templates := "SrcType := Byte" } EQ_Contact(in1 := "4号梯数据块"."4号梯当前楼层", in2 := 10)
      Coil( "4号梯数据块"."4号梯10层flag" )
   END_RUNG
   // the same network as SCL:
   "4号梯数据块"."4号梯1层flag" := "4号梯数据块"."4号梯当前楼层" = 1;
   "4号梯数据块"."4号梯2层flag" := "4号梯数据块"."4号梯当前楼层" = 2;
   "4号梯数据块"."4号梯3层flag" := "4号梯数据块"."4号梯当前楼层" = 3;
   "4号梯数据块"."4号梯4层flag" := "4号梯数据块"."4号梯当前楼层" = 4;
   "4号梯数据块"."4号梯5层flag" := "4号梯数据块"."4号梯当前楼层" = 5;
   "4号梯数据块"."4号梯6层flag" := "4号梯数据块"."4号梯当前楼层" = 6;
   "4号梯数据块"."4号梯7层flag" := "4号梯数据块"."4号梯当前楼层" = 7;
   "4号梯数据块"."4号梯8层flag" := "4号梯数据块"."4号梯当前楼层" = 8;
   "4号梯数据块"."4号梯9层flag" := "4号梯数据块"."4号梯当前楼层" = 9;
   "4号梯数据块"."4号梯10层flag" := "4号梯数据块"."4号梯当前楼层" = 10;
END_REGION

REGION Network 2: 4号梯楼层led_a显示
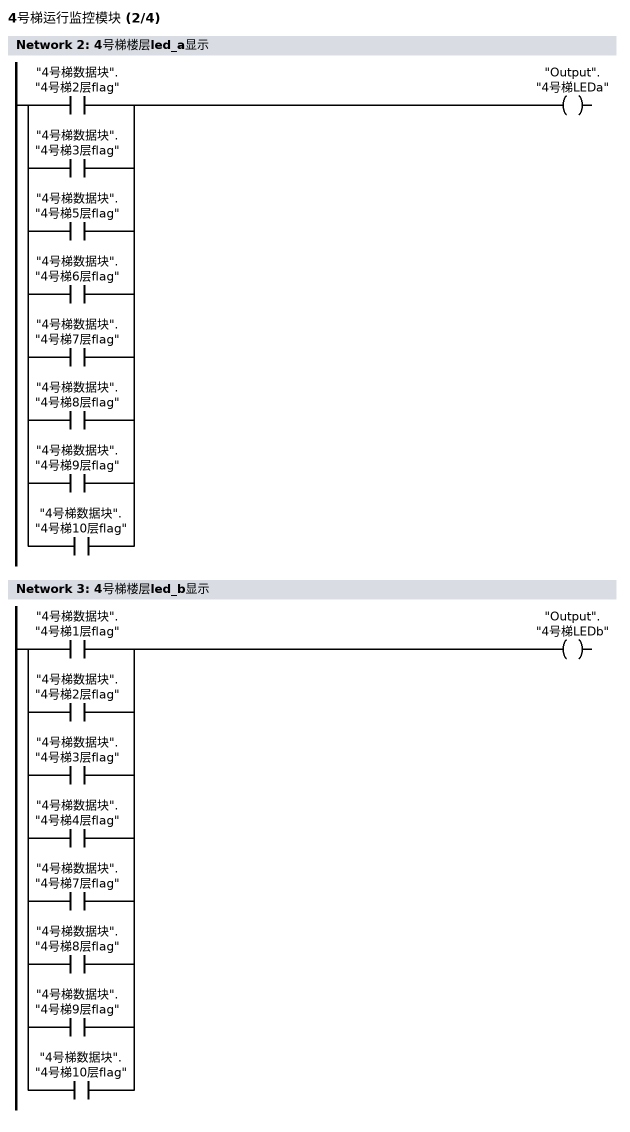
   RUNG wire#powerrail
      Contact( "4号梯数据块"."4号梯2层flag" )
      wire#w1
      Coil( "Output"."4号梯LEDa" )
   END_RUNG
   RUNG wire#powerrail
      Contact( "4号梯数据块"."4号梯3层flag" )
   END_RUNG wire#w1
   RUNG wire#powerrail
      Contact( "4号梯数据块"."4号梯5层flag" )
   END_RUNG wire#w1
   RUNG wire#powerrail
      Contact( "4号梯数据块"."4号梯6层flag" )
   END_RUNG wire#w1
   RUNG wire#powerrail
      Contact( "4号梯数据块"."4号梯7层flag" )
   END_RUNG wire#w1
   RUNG wire#powerrail
      Contact( "4号梯数据块"."4号梯8层flag" )
   END_RUNG wire#w1
   RUNG wire#powerrail
      Contact( "4号梯数据块"."4号梯9层flag" )
   END_RUNG wire#w1
   RUNG wire#powerrail
      Contact( "4号梯数据块"."4号梯10层flag" )
   END_RUNG wire#w1
   // the same network as SCL:
   "Output"."4号梯LEDa" := "4号梯数据块"."4号梯2层flag" OR "4号梯数据块"."4号梯3层flag" OR "4号梯数据块"."4号梯5层flag" OR "4号梯数据块"."4号梯6层flag" OR "4号梯数据块"."4号梯7层flag" OR "4号梯数据块"."4号梯8层flag" OR "4号梯数据块"."4号梯9层flag" OR "4号梯数据块"."4号梯10层flag";
END_REGION

REGION Network 3: 4号梯楼层led_b显示
   RUNG wire#powerrail
      Contact( "4号梯数据块"."4号梯1层flag" )
      wire#w1
      Coil( "Output"."4号梯LEDb" )
   END_RUNG
   RUNG wire#powerrail
      Contact( "4号梯数据块"."4号梯2层flag" )
   END_RUNG wire#w1
   RUNG wire#powerrail
      Contact( "4号梯数据块"."4号梯3层flag" )
   END_RUNG wire#w1
   RUNG wire#powerrail
      Contact( "4号梯数据块"."4号梯4层flag" )
   END_RUNG wire#w1
   RUNG wire#powerrail
      Contact( "4号梯数据块"."4号梯7层flag" )
   END_RUNG wire#w1
   RUNG wire#powerrail
      Contact( "4号梯数据块"."4号梯8层flag" )
   END_RUNG wire#w1
   RUNG wire#powerrail
      Contact( "4号梯数据块"."4号梯9层flag" )
   END_RUNG wire#w1
   RUNG wire#powerrail
      Contact( "4号梯数据块"."4号梯10层flag" )
   END_RUNG wire#w1
   // the same network as SCL:
   "Output"."4号梯LEDb" := "4号梯数据块"."4号梯1层flag" OR "4号梯数据块"."4号梯2层flag" OR "4号梯数据块"."4号梯3层flag" OR "4号梯数据块"."4号梯4层flag" OR "4号梯数据块"."4号梯7层flag" OR "4号梯数据块"."4号梯8层flag" OR "4号梯数据块"."4号梯9层flag" OR "4号梯数据块"."4号梯10层flag";
END_REGION

REGION Network 4: 4号梯楼层led_c显示
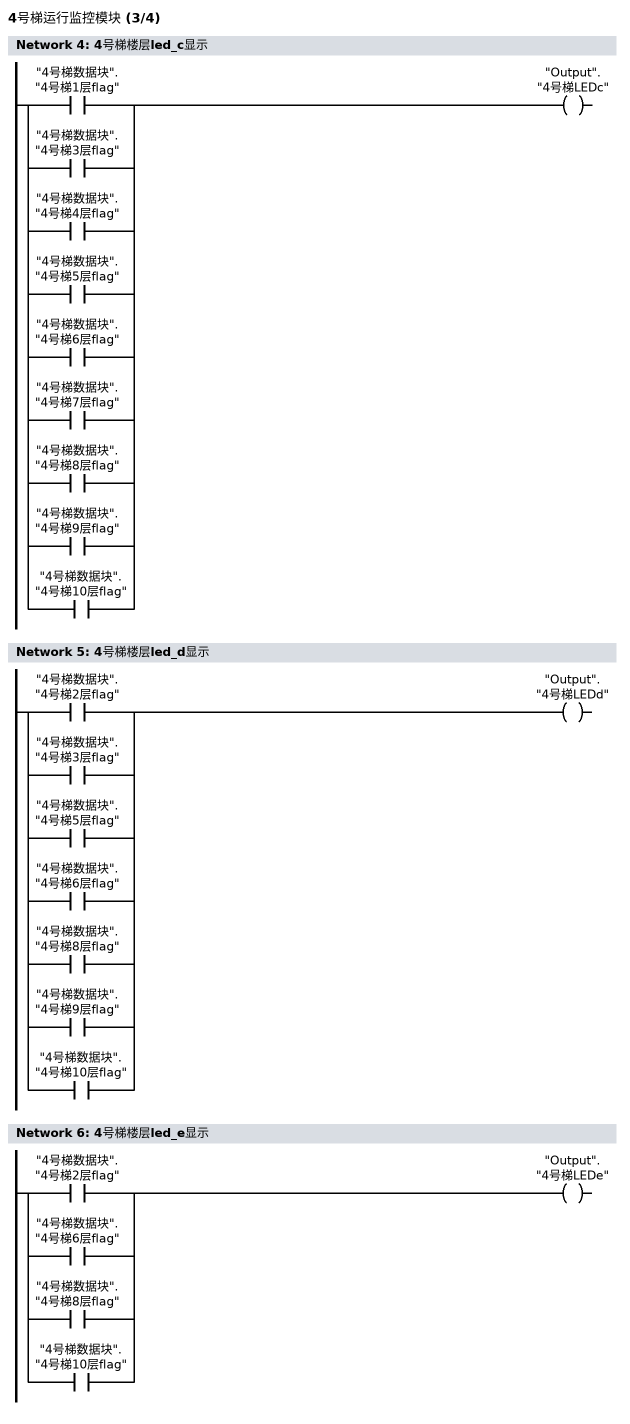
   RUNG wire#powerrail
      Contact( "4号梯数据块"."4号梯1层flag" )
      wire#w1
      Coil( "Output"."4号梯LEDc" )
   END_RUNG
   RUNG wire#powerrail
      Contact( "4号梯数据块"."4号梯3层flag" )
   END_RUNG wire#w1
   RUNG wire#powerrail
      Contact( "4号梯数据块"."4号梯4层flag" )
   END_RUNG wire#w1
   RUNG wire#powerrail
      Contact( "4号梯数据块"."4号梯5层flag" )
   END_RUNG wire#w1
   RUNG wire#powerrail
      Contact( "4号梯数据块"."4号梯6层flag" )
   END_RUNG wire#w1
   RUNG wire#powerrail
      Contact( "4号梯数据块"."4号梯7层flag" )
   END_RUNG wire#w1
   RUNG wire#powerrail
      Contact( "4号梯数据块"."4号梯8层flag" )
   END_RUNG wire#w1
   RUNG wire#powerrail
      Contact( "4号梯数据块"."4号梯9层flag" )
   END_RUNG wire#w1
   RUNG wire#powerrail
      Contact( "4号梯数据块"."4号梯10层flag" )
   END_RUNG wire#w1
   // the same network as SCL:
   "Output"."4号梯LEDc" := "4号梯数据块"."4号梯1层flag" OR "4号梯数据块"."4号梯3层flag" OR "4号梯数据块"."4号梯4层flag" OR "4号梯数据块"."4号梯5层flag" OR "4号梯数据块"."4号梯6层flag" OR "4号梯数据块"."4号梯7层flag" OR "4号梯数据块"."4号梯8层flag" OR "4号梯数据块"."4号梯9层flag" OR "4号梯数据块"."4号梯10层flag";
END_REGION

REGION Network 5: 4号梯楼层led_d显示
   RUNG wire#powerrail
      Contact( "4号梯数据块"."4号梯2层flag" )
      wire#w1
      Coil( "Output"."4号梯LEDd" )
   END_RUNG
   RUNG wire#powerrail
      Contact( "4号梯数据块"."4号梯3层flag" )
   END_RUNG wire#w1
   RUNG wire#powerrail
      Contact( "4号梯数据块"."4号梯5层flag" )
   END_RUNG wire#w1
   RUNG wire#powerrail
      Contact( "4号梯数据块"."4号梯6层flag" )
   END_RUNG wire#w1
   RUNG wire#powerrail
      Contact( "4号梯数据块"."4号梯8层flag" )
   END_RUNG wire#w1
   RUNG wire#powerrail
      Contact( "4号梯数据块"."4号梯9层flag" )
   END_RUNG wire#w1
   RUNG wire#powerrail
      Contact( "4号梯数据块"."4号梯10层flag" )
   END_RUNG wire#w1
   // the same network as SCL:
   "Output"."4号梯LEDd" := "4号梯数据块"."4号梯2层flag" OR "4号梯数据块"."4号梯3层flag" OR "4号梯数据块"."4号梯5层flag" OR "4号梯数据块"."4号梯6层flag" OR "4号梯数据块"."4号梯8层flag" OR "4号梯数据块"."4号梯9层flag" OR "4号梯数据块"."4号梯10层flag";
END_REGION

REGION Network 6: 4号梯楼层led_e显示
   RUNG wire#powerrail
      Contact( "4号梯数据块"."4号梯2层flag" )
      wire#w1
      Coil( "Output"."4号梯LEDe" )
   END_RUNG
   RUNG wire#powerrail
      Contact( "4号梯数据块"."4号梯6层flag" )
   END_RUNG wire#w1
   RUNG wire#powerrail
      Contact( "4号梯数据块"."4号梯8层flag" )
   END_RUNG wire#w1
   RUNG wire#powerrail
      Contact( "4号梯数据块"."4号梯10层flag" )
   END_RUNG wire#w1
   // the same network as SCL:
   "Output"."4号梯LEDe" := "4号梯数据块"."4号梯2层flag" OR "4号梯数据块"."4号梯6层flag" OR "4号梯数据块"."4号梯8层flag" OR "4号梯数据块"."4号梯10层flag";
END_REGION

REGION Network 7: 4号梯楼层led_f显示
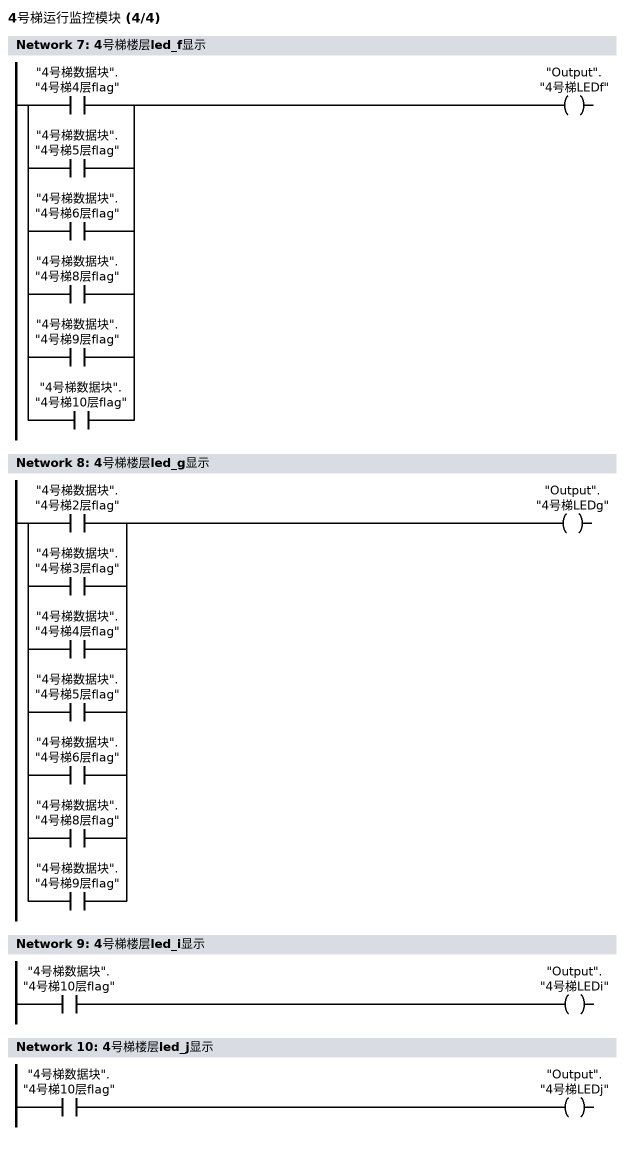
   RUNG wire#powerrail
      Contact( "4号梯数据块"."4号梯4层flag" )
      wire#w1
      Coil( "Output"."4号梯LEDf" )
   END_RUNG
   RUNG wire#powerrail
      Contact( "4号梯数据块"."4号梯5层flag" )
   END_RUNG wire#w1
   RUNG wire#powerrail
      Contact( "4号梯数据块"."4号梯6层flag" )
   END_RUNG wire#w1
   RUNG wire#powerrail
      Contact( "4号梯数据块"."4号梯8层flag" )
   END_RUNG wire#w1
   RUNG wire#powerrail
      Contact( "4号梯数据块"."4号梯9层flag" )
   END_RUNG wire#w1
   RUNG wire#powerrail
      Contact( "4号梯数据块"."4号梯10层flag" )
   END_RUNG wire#w1
   // the same network as SCL:
   "Output"."4号梯LEDf" := "4号梯数据块"."4号梯4层flag" OR "4号梯数据块"."4号梯5层flag" OR "4号梯数据块"."4号梯6层flag" OR "4号梯数据块"."4号梯8层flag" OR "4号梯数据块"."4号梯9层flag" OR "4号梯数据块"."4号梯10层flag";
END_REGION

REGION Network 8: 4号梯楼层led_g显示
   RUNG wire#powerrail
      Contact( "4号梯数据块"."4号梯2层flag" )
      wire#w1
      Coil( "Output"."4号梯LEDg" )
   END_RUNG
   RUNG wire#powerrail
      Contact( "4号梯数据块"."4号梯3层flag" )
   END_RUNG wire#w1
   RUNG wire#powerrail
      Contact( "4号梯数据块"."4号梯4层flag" )
   END_RUNG wire#w1
   RUNG wire#powerrail
      Contact( "4号梯数据块"."4号梯5层flag" )
   END_RUNG wire#w1
   RUNG wire#powerrail
      Contact( "4号梯数据块"."4号梯6层flag" )
   END_RUNG wire#w1
   RUNG wire#powerrail
      Contact( "4号梯数据块"."4号梯8层flag" )
   END_RUNG wire#w1
   RUNG wire#powerrail
      Contact( "4号梯数据块"."4号梯9层flag" )
   END_RUNG wire#w1
   // the same network as SCL:
   "Output"."4号梯LEDg" := "4号梯数据块"."4号梯2层flag" OR "4号梯数据块"."4号梯3层flag" OR "4号梯数据块"."4号梯4层flag" OR "4号梯数据块"."4号梯5层flag" OR "4号梯数据块"."4号梯6层flag" OR "4号梯数据块"."4号梯8层flag" OR "4号梯数据块"."4号梯9层flag";
END_REGION

REGION Network 9: 4号梯楼层led_i显示
   RUNG wire#powerrail
      Contact( "4号梯数据块"."4号梯10层flag" )
      Coil( "Output"."4号梯LEDi" )
   END_RUNG
   // the same network as SCL:
   "Output"."4号梯LEDi" := "4号梯数据块"."4号梯10层flag";
END_REGION

REGION Network 10: 4号梯楼层led_j显示
   RUNG wire#powerrail
      Contact( "4号梯数据块"."4号梯10层flag" )
      Coil( "Output"."4号梯LEDj" )
   END_RUNG
   // the same network as SCL:
   "Output"."4号梯LEDj" := "4号梯数据块"."4号梯10层flag";
END_REGION
END_FUNCTION

FUNCTION "4号梯检修" : Void   // FC22, LAD
{ S7_Optimized_Access := 'TRUE' }
VERSION : 0.1
BEGIN
END_FUNCTION

FUNCTION "4号梯超重与内选" : Void   // FC23, LAD
{ S7_Optimized_Access := 'TRUE' }
VERSION : 0.1
BEGIN
END_FUNCTION

FUNCTION "4号梯开关门控制" : Void   // FC29, LAD
{ S7_Optimized_Access := 'TRUE' }
VERSION : 0.1
BEGIN
END_FUNCTION

FUNCTION "4号梯楼层计数" : Void   // FC35, LAD
{ S7_Optimized_Access := 'TRUE' }
VERSION : 0.1
BEGIN
END_FUNCTION

FUNCTION "4号梯目标楼层与方向判断" : Void   // FC51, LAD
{ S7_Optimized_Access := 'TRUE' }
VERSION : 0.1
BEGIN
END_FUNCTION

FUNCTION "4号梯字节消除与记录" : Void   // FC52, LAD
{ S7_Optimized_Access := 'TRUE' }
VERSION : 0.1
BEGIN
END_FUNCTION

FUNCTION "4号梯启停控制" : Void   // FC61, LAD
{ S7_Optimized_Access := 'TRUE' }
VERSION : 0.1
BEGIN
END_FUNCTION

// folder: 5号梯

FUNCTION "5号梯主函数" : Void   // FC2, LAD
{ S7_Optimized_Access := 'TRUE' }
VERSION : 0.1
BEGIN

REGION Network 1
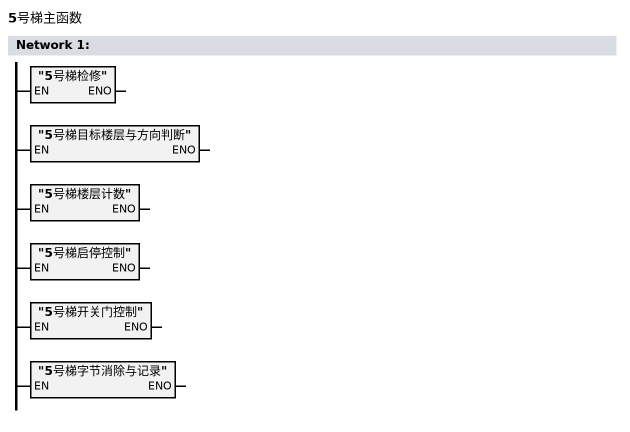
   RUNG wire#powerrail
      "5号梯检修"()
   END_RUNG
   RUNG wire#powerrail
      "5号梯目标楼层与方向判断"()
   END_RUNG
   RUNG wire#powerrail
      "5号梯楼层计数"()
   END_RUNG
   RUNG wire#powerrail
      "5号梯启停控制"()
   END_RUNG
   RUNG wire#powerrail
      "5号梯开关门控制"()
   END_RUNG
   RUNG wire#powerrail
      "5号梯字节消除与记录"()
   END_RUNG
   // the same network as SCL:
   "5号梯检修"();
   "5号梯目标楼层与方向判断"();
   "5号梯楼层计数"();
   "5号梯启停控制"();
   "5号梯开关门控制"();
   "5号梯字节消除与记录"();
END_REGION
END_FUNCTION

FUNCTION "5号梯初始化" : Void   // FC6, LAD
{ S7_Optimized_Access := 'TRUE' }
VERSION : 0.1
   VAR_INPUT
      初始化方向 : Bool;
      初始化楼层 : Byte;
   END_VAR
   VAR_TEMP   // added for the SCL form of the ladder/FBD networks
      _w1 : Bool;
      _w2 : Bool;
      _w3 : Bool;
      _w4 : Bool;
   END_VAR
BEGIN

REGION Network 1: 5号梯传参（方向+初始化楼层）
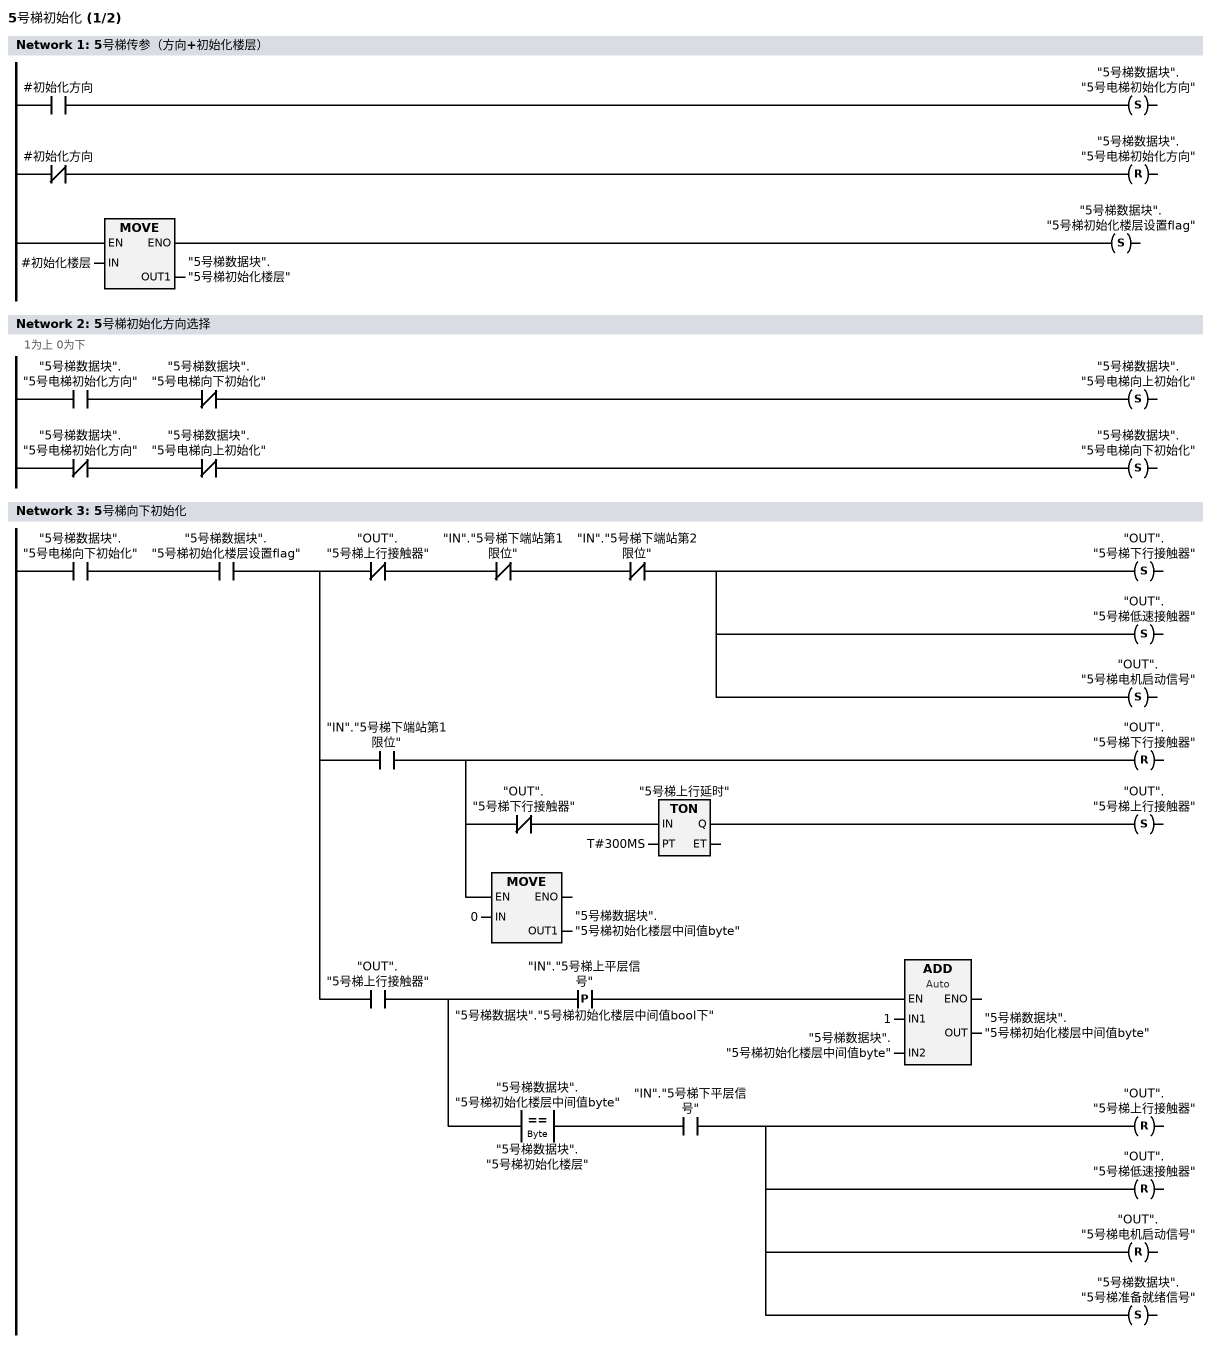
   RUNG wire#powerrail
      Contact( #初始化方向 )
      S_Coil( "5号梯数据块"."5号电梯初始化方向" )
   END_RUNG
   RUNG wire#powerrail
      I_Contact( #初始化方向 )
      R_Coil( "5号梯数据块"."5号电梯初始化方向" )
   END_RUNG
   RUNG wire#powerrail
      Move(in := #初始化楼层, out1 => "5号梯数据块"."5号梯初始化楼层")
      S_Coil( "5号梯数据块"."5号梯初始化楼层设置flag" )
   END_RUNG
   // the same network as SCL:
   IF #初始化方向 THEN "5号梯数据块"."5号电梯初始化方向" := TRUE; END_IF;
   IF NOT #初始化方向 THEN "5号梯数据块"."5号电梯初始化方向" := FALSE; END_IF;
   "5号梯数据块"."5号梯初始化楼层" := #初始化楼层;
   "5号梯数据块"."5号梯初始化楼层设置flag" := TRUE;
END_REGION

REGION Network 2: 5号梯初始化方向选择
   // 1为上 0为下
   RUNG wire#powerrail
      Contact( "5号梯数据块"."5号电梯初始化方向" )
      I_Contact( "5号梯数据块"."5号电梯向下初始化" )
      S_Coil( "5号梯数据块"."5号电梯向上初始化" )
   END_RUNG
   RUNG wire#powerrail
      I_Contact( "5号梯数据块"."5号电梯初始化方向" )
      I_Contact( "5号梯数据块"."5号电梯向上初始化" )
      S_Coil( "5号梯数据块"."5号电梯向下初始化" )
   END_RUNG
   // the same network as SCL:
   IF "5号梯数据块"."5号电梯初始化方向" AND NOT "5号梯数据块"."5号电梯向下初始化" THEN "5号梯数据块"."5号电梯向上初始化" := TRUE; END_IF;
   IF NOT "5号梯数据块"."5号电梯初始化方向" AND NOT "5号梯数据块"."5号电梯向上初始化" THEN "5号梯数据块"."5号电梯向下初始化" := TRUE; END_IF;
END_REGION

REGION Network 3: 5号梯向下初始化
   #_w1 := "5号梯数据块"."5号电梯向下初始化" AND "5号梯数据块"."5号梯初始化楼层设置flag";
   IF #_w1 AND NOT "OUT"."5号梯上行接触器" AND NOT "IN"."5号梯下端站第1限位" AND NOT "IN"."5号梯下端站第2限位" THEN
       "OUT"."5号梯下行接触器" := TRUE;
       "OUT"."5号梯低速接触器" := TRUE;
       "OUT"."5号梯电机启动信号" := TRUE;
   END_IF;
   #_w2 := #_w1 AND "IN"."5号梯下端站第1限位";
   IF #_w2 THEN "OUT"."5号梯下行接触器" := FALSE; END_IF;
   "5号梯上行延时".TON(IN := #_w2 AND NOT "OUT"."5号梯下行接触器", PT := T#300MS);
   IF "5号梯上行延时".Q THEN "OUT"."5号梯上行接触器" := TRUE; END_IF;
   IF #_w2 THEN "5号梯数据块"."5号梯初始化楼层中间值byte" := 0; END_IF;
   #_w3 := #_w1 AND "OUT"."5号梯上行接触器";
   #_w4 := #_w3 AND "IN"."5号梯上平层信号" AND NOT "5号梯数据块"."5号梯初始化楼层中间值bool下";   // rising edge of "IN"."5号梯上平层信号"
   "5号梯数据块"."5号梯初始化楼层中间值bool下" := "IN"."5号梯上平层信号";
   IF #_w4 THEN "5号梯数据块"."5号梯初始化楼层中间值byte" := 1 + "5号梯数据块"."5号梯初始化楼层中间值byte"; END_IF;
   IF #_w3 AND ("5号梯数据块"."5号梯初始化楼层中间值byte" = "5号梯数据块"."5号梯初始化楼层") AND "IN"."5号梯下平层信号" THEN
       "OUT"."5号梯上行接触器" := FALSE;
       "OUT"."5号梯低速接触器" := FALSE;
       "OUT"."5号梯电机启动信号" := FALSE;
       "5号梯数据块"."5号梯准备就绪信号" := TRUE;
   END_IF;
END_REGION

REGION Network 4: 5号梯向上初始化
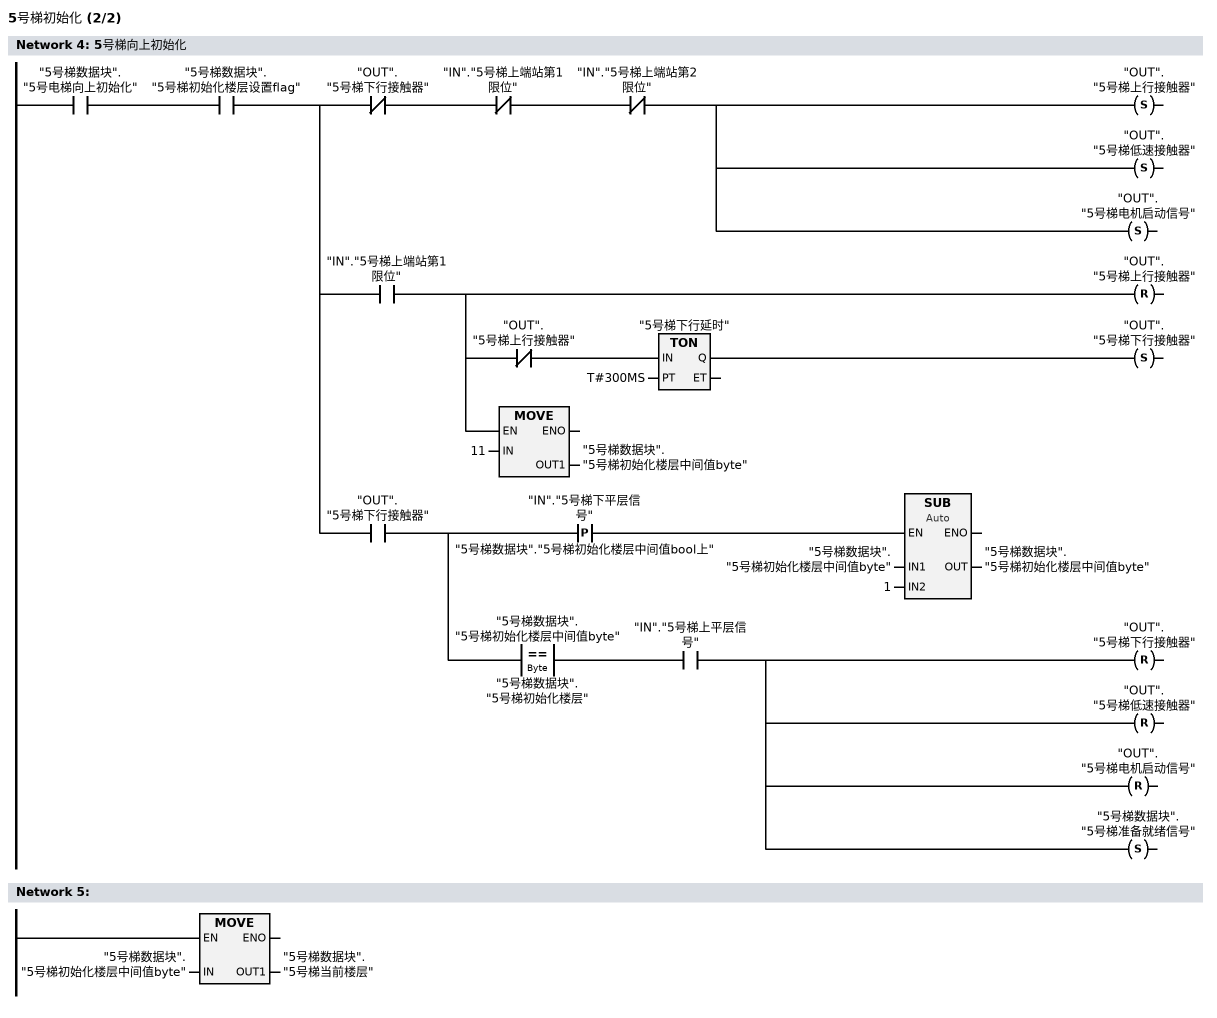
   #_w1 := "5号梯数据块"."5号电梯向上初始化" AND "5号梯数据块"."5号梯初始化楼层设置flag";
   IF #_w1 AND NOT "OUT"."5号梯下行接触器" AND NOT "IN"."5号梯上端站第1限位" AND NOT "IN"."5号梯上端站第2限位" THEN
       "OUT"."5号梯上行接触器" := TRUE;
       "OUT"."5号梯低速接触器" := TRUE;
       "OUT"."5号梯电机启动信号" := TRUE;
   END_IF;
   #_w2 := #_w1 AND "IN"."5号梯上端站第1限位";
   IF #_w2 THEN "OUT"."5号梯上行接触器" := FALSE; END_IF;
   "5号梯下行延时".TON(IN := #_w2 AND NOT "OUT"."5号梯上行接触器", PT := T#300MS);
   IF "5号梯下行延时".Q THEN "OUT"."5号梯下行接触器" := TRUE; END_IF;
   IF #_w2 THEN "5号梯数据块"."5号梯初始化楼层中间值byte" := 11; END_IF;
   #_w3 := #_w1 AND "OUT"."5号梯下行接触器";
   #_w4 := #_w3 AND "IN"."5号梯下平层信号" AND NOT "5号梯数据块"."5号梯初始化楼层中间值bool上";   // rising edge of "IN"."5号梯下平层信号"
   "5号梯数据块"."5号梯初始化楼层中间值bool上" := "IN"."5号梯下平层信号";
   IF #_w4 THEN "5号梯数据块"."5号梯初始化楼层中间值byte" := "5号梯数据块"."5号梯初始化楼层中间值byte" - 1; END_IF;
   IF #_w3 AND ("5号梯数据块"."5号梯初始化楼层中间值byte" = "5号梯数据块"."5号梯初始化楼层") AND "IN"."5号梯上平层信号" THEN
       "OUT"."5号梯下行接触器" := FALSE;
       "OUT"."5号梯低速接触器" := FALSE;
       "OUT"."5号梯电机启动信号" := FALSE;
       "5号梯数据块"."5号梯准备就绪信号" := TRUE;
   END_IF;
END_REGION

REGION Network 5
   RUNG wire#powerrail
      Move(in := "5号梯数据块"."5号梯初始化楼层中间值byte", out1 => "5号梯数据块"."5号梯当前楼层")
   END_RUNG
   // the same network as SCL:
   "5号梯数据块"."5号梯当前楼层" := "5号梯数据块"."5号梯初始化楼层中间值byte";
END_REGION
END_FUNCTION

FUNCTION "5号梯运行监控模块" : Void   // FC18, LAD
{ S7_Optimized_Access := 'TRUE' }
VERSION : 0.1
BEGIN

REGION Network 1: 5号梯获取当前楼层设置标志位
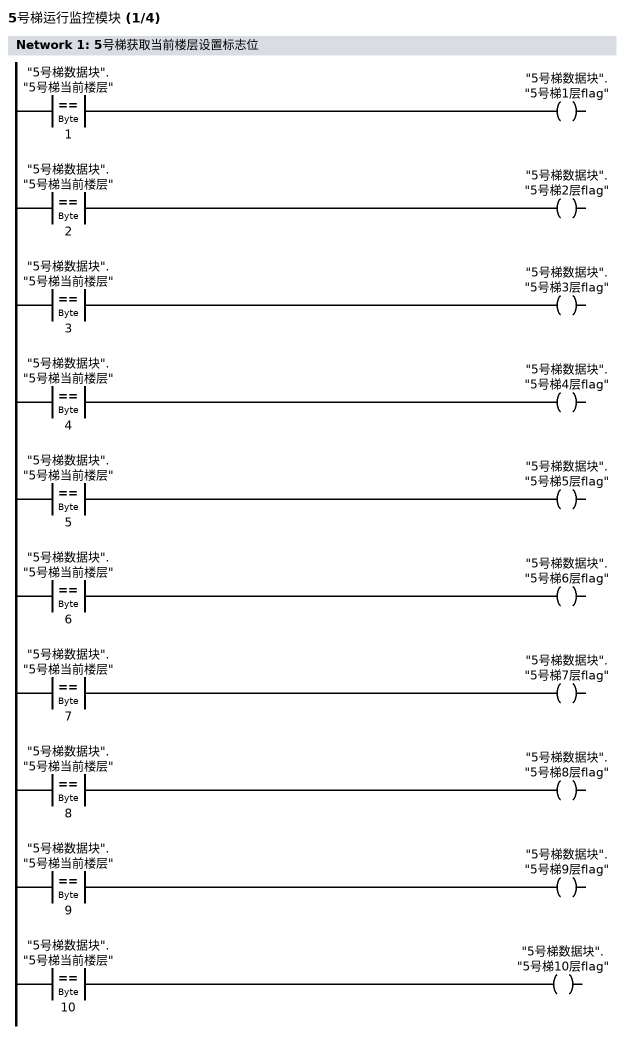
   RUNG wire#powerrail
      { S7_Templates := "SrcType := Byte" } EQ_Contact(in1 := "5号梯数据块"."5号梯当前楼层", in2 := 1)
      Coil( "5号梯数据块"."5号梯1层flag" )
   END_RUNG
   RUNG wire#powerrail
      { S7_Templates := "SrcType := Byte" } EQ_Contact(in1 := "5号梯数据块"."5号梯当前楼层", in2 := 2)
      Coil( "5号梯数据块"."5号梯2层flag" )
   END_RUNG
   RUNG wire#powerrail
      { S7_Templates := "SrcType := Byte" } EQ_Contact(in1 := "5号梯数据块"."5号梯当前楼层", in2 := 3)
      Coil( "5号梯数据块"."5号梯3层flag" )
   END_RUNG
   RUNG wire#powerrail
      { S7_Templates := "SrcType := Byte" } EQ_Contact(in1 := "5号梯数据块"."5号梯当前楼层", in2 := 4)
      Coil( "5号梯数据块"."5号梯4层flag" )
   END_RUNG
   RUNG wire#powerrail
      { S7_Templates := "SrcType := Byte" } EQ_Contact(in1 := "5号梯数据块"."5号梯当前楼层", in2 := 5)
      Coil( "5号梯数据块"."5号梯5层flag" )
   END_RUNG
   RUNG wire#powerrail
      { S7_Templates := "SrcType := Byte" } EQ_Contact(in1 := "5号梯数据块"."5号梯当前楼层", in2 := 6)
      Coil( "5号梯数据块"."5号梯6层flag" )
   END_RUNG
   RUNG wire#powerrail
      { S7_Templates := "SrcType := Byte" } EQ_Contact(in1 := "5号梯数据块"."5号梯当前楼层", in2 := 7)
      Coil( "5号梯数据块"."5号梯7层flag" )
   END_RUNG
   RUNG wire#powerrail
      { S7_Templates := "SrcType := Byte" } EQ_Contact(in1 := "5号梯数据块"."5号梯当前楼层", in2 := 8)
      Coil( "5号梯数据块"."5号梯8层flag" )
   END_RUNG
   RUNG wire#powerrail
      { S7_Templates := "SrcType := Byte" } EQ_Contact(in1 := "5号梯数据块"."5号梯当前楼层", in2 := 9)
      Coil( "5号梯数据块"."5号梯9层flag" )
   END_RUNG
   RUNG wire#powerrail
      { S7_Templates := "SrcType := Byte" } EQ_Contact(in1 := "5号梯数据块"."5号梯当前楼层", in2 := 10)
      Coil( "5号梯数据块"."5号梯10层flag" )
   END_RUNG
   // the same network as SCL:
   "5号梯数据块"."5号梯1层flag" := "5号梯数据块"."5号梯当前楼层" = 1;
   "5号梯数据块"."5号梯2层flag" := "5号梯数据块"."5号梯当前楼层" = 2;
   "5号梯数据块"."5号梯3层flag" := "5号梯数据块"."5号梯当前楼层" = 3;
   "5号梯数据块"."5号梯4层flag" := "5号梯数据块"."5号梯当前楼层" = 4;
   "5号梯数据块"."5号梯5层flag" := "5号梯数据块"."5号梯当前楼层" = 5;
   "5号梯数据块"."5号梯6层flag" := "5号梯数据块"."5号梯当前楼层" = 6;
   "5号梯数据块"."5号梯7层flag" := "5号梯数据块"."5号梯当前楼层" = 7;
   "5号梯数据块"."5号梯8层flag" := "5号梯数据块"."5号梯当前楼层" = 8;
   "5号梯数据块"."5号梯9层flag" := "5号梯数据块"."5号梯当前楼层" = 9;
   "5号梯数据块"."5号梯10层flag" := "5号梯数据块"."5号梯当前楼层" = 10;
END_REGION

REGION Network 2: 5号梯楼层led_a显示
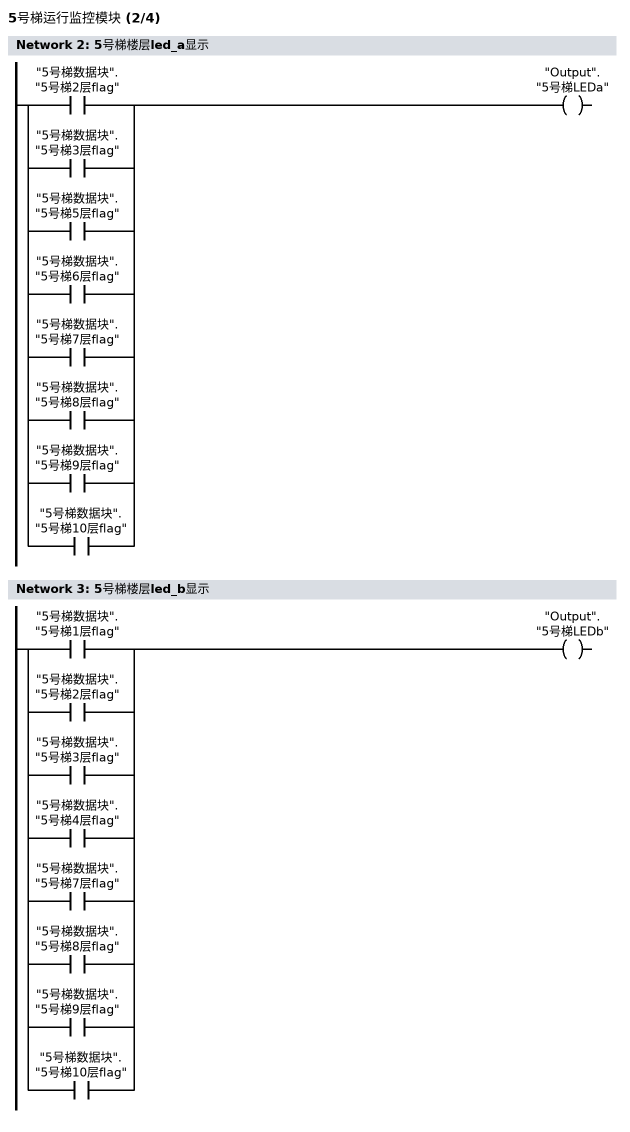
   RUNG wire#powerrail
      Contact( "5号梯数据块"."5号梯2层flag" )
      wire#w1
      Coil( "Output"."5号梯LEDa" )
   END_RUNG
   RUNG wire#powerrail
      Contact( "5号梯数据块"."5号梯3层flag" )
   END_RUNG wire#w1
   RUNG wire#powerrail
      Contact( "5号梯数据块"."5号梯5层flag" )
   END_RUNG wire#w1
   RUNG wire#powerrail
      Contact( "5号梯数据块"."5号梯6层flag" )
   END_RUNG wire#w1
   RUNG wire#powerrail
      Contact( "5号梯数据块"."5号梯7层flag" )
   END_RUNG wire#w1
   RUNG wire#powerrail
      Contact( "5号梯数据块"."5号梯8层flag" )
   END_RUNG wire#w1
   RUNG wire#powerrail
      Contact( "5号梯数据块"."5号梯9层flag" )
   END_RUNG wire#w1
   RUNG wire#powerrail
      Contact( "5号梯数据块"."5号梯10层flag" )
   END_RUNG wire#w1
   // the same network as SCL:
   "Output"."5号梯LEDa" := "5号梯数据块"."5号梯2层flag" OR "5号梯数据块"."5号梯3层flag" OR "5号梯数据块"."5号梯5层flag" OR "5号梯数据块"."5号梯6层flag" OR "5号梯数据块"."5号梯7层flag" OR "5号梯数据块"."5号梯8层flag" OR "5号梯数据块"."5号梯9层flag" OR "5号梯数据块"."5号梯10层flag";
END_REGION

REGION Network 3: 5号梯楼层led_b显示
   RUNG wire#powerrail
      Contact( "5号梯数据块"."5号梯1层flag" )
      wire#w1
      Coil( "Output"."5号梯LEDb" )
   END_RUNG
   RUNG wire#powerrail
      Contact( "5号梯数据块"."5号梯2层flag" )
   END_RUNG wire#w1
   RUNG wire#powerrail
      Contact( "5号梯数据块"."5号梯3层flag" )
   END_RUNG wire#w1
   RUNG wire#powerrail
      Contact( "5号梯数据块"."5号梯4层flag" )
   END_RUNG wire#w1
   RUNG wire#powerrail
      Contact( "5号梯数据块"."5号梯7层flag" )
   END_RUNG wire#w1
   RUNG wire#powerrail
      Contact( "5号梯数据块"."5号梯8层flag" )
   END_RUNG wire#w1
   RUNG wire#powerrail
      Contact( "5号梯数据块"."5号梯9层flag" )
   END_RUNG wire#w1
   RUNG wire#powerrail
      Contact( "5号梯数据块"."5号梯10层flag" )
   END_RUNG wire#w1
   // the same network as SCL:
   "Output"."5号梯LEDb" := "5号梯数据块"."5号梯1层flag" OR "5号梯数据块"."5号梯2层flag" OR "5号梯数据块"."5号梯3层flag" OR "5号梯数据块"."5号梯4层flag" OR "5号梯数据块"."5号梯7层flag" OR "5号梯数据块"."5号梯8层flag" OR "5号梯数据块"."5号梯9层flag" OR "5号梯数据块"."5号梯10层flag";
END_REGION

REGION Network 4: 5号梯楼层led_c显示
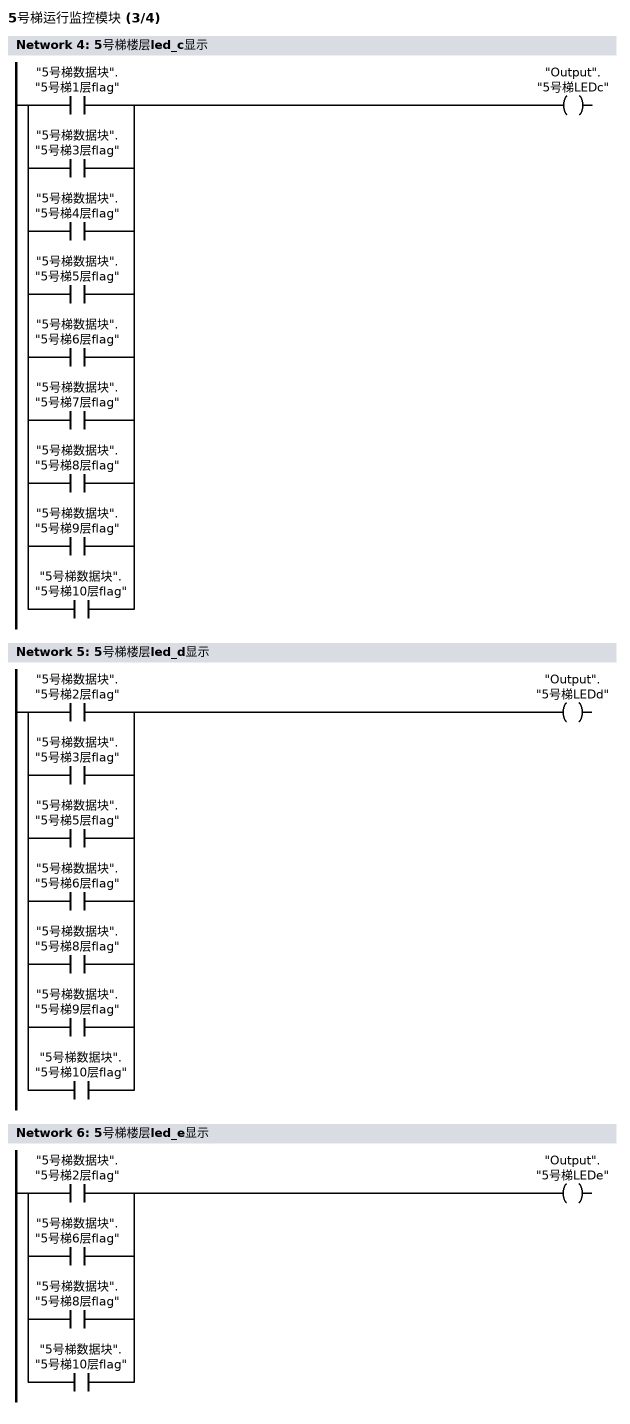
   RUNG wire#powerrail
      Contact( "5号梯数据块"."5号梯1层flag" )
      wire#w1
      Coil( "Output"."5号梯LEDc" )
   END_RUNG
   RUNG wire#powerrail
      Contact( "5号梯数据块"."5号梯3层flag" )
   END_RUNG wire#w1
   RUNG wire#powerrail
      Contact( "5号梯数据块"."5号梯4层flag" )
   END_RUNG wire#w1
   RUNG wire#powerrail
      Contact( "5号梯数据块"."5号梯5层flag" )
   END_RUNG wire#w1
   RUNG wire#powerrail
      Contact( "5号梯数据块"."5号梯6层flag" )
   END_RUNG wire#w1
   RUNG wire#powerrail
      Contact( "5号梯数据块"."5号梯7层flag" )
   END_RUNG wire#w1
   RUNG wire#powerrail
      Contact( "5号梯数据块"."5号梯8层flag" )
   END_RUNG wire#w1
   RUNG wire#powerrail
      Contact( "5号梯数据块"."5号梯9层flag" )
   END_RUNG wire#w1
   RUNG wire#powerrail
      Contact( "5号梯数据块"."5号梯10层flag" )
   END_RUNG wire#w1
   // the same network as SCL:
   "Output"."5号梯LEDc" := "5号梯数据块"."5号梯1层flag" OR "5号梯数据块"."5号梯3层flag" OR "5号梯数据块"."5号梯4层flag" OR "5号梯数据块"."5号梯5层flag" OR "5号梯数据块"."5号梯6层flag" OR "5号梯数据块"."5号梯7层flag" OR "5号梯数据块"."5号梯8层flag" OR "5号梯数据块"."5号梯9层flag" OR "5号梯数据块"."5号梯10层flag";
END_REGION

REGION Network 5: 5号梯楼层led_d显示
   RUNG wire#powerrail
      Contact( "5号梯数据块"."5号梯2层flag" )
      wire#w1
      Coil( "Output"."5号梯LEDd" )
   END_RUNG
   RUNG wire#powerrail
      Contact( "5号梯数据块"."5号梯3层flag" )
   END_RUNG wire#w1
   RUNG wire#powerrail
      Contact( "5号梯数据块"."5号梯5层flag" )
   END_RUNG wire#w1
   RUNG wire#powerrail
      Contact( "5号梯数据块"."5号梯6层flag" )
   END_RUNG wire#w1
   RUNG wire#powerrail
      Contact( "5号梯数据块"."5号梯8层flag" )
   END_RUNG wire#w1
   RUNG wire#powerrail
      Contact( "5号梯数据块"."5号梯9层flag" )
   END_RUNG wire#w1
   RUNG wire#powerrail
      Contact( "5号梯数据块"."5号梯10层flag" )
   END_RUNG wire#w1
   // the same network as SCL:
   "Output"."5号梯LEDd" := "5号梯数据块"."5号梯2层flag" OR "5号梯数据块"."5号梯3层flag" OR "5号梯数据块"."5号梯5层flag" OR "5号梯数据块"."5号梯6层flag" OR "5号梯数据块"."5号梯8层flag" OR "5号梯数据块"."5号梯9层flag" OR "5号梯数据块"."5号梯10层flag";
END_REGION

REGION Network 6: 5号梯楼层led_e显示
   RUNG wire#powerrail
      Contact( "5号梯数据块"."5号梯2层flag" )
      wire#w1
      Coil( "Output"."5号梯LEDe" )
   END_RUNG
   RUNG wire#powerrail
      Contact( "5号梯数据块"."5号梯6层flag" )
   END_RUNG wire#w1
   RUNG wire#powerrail
      Contact( "5号梯数据块"."5号梯8层flag" )
   END_RUNG wire#w1
   RUNG wire#powerrail
      Contact( "5号梯数据块"."5号梯10层flag" )
   END_RUNG wire#w1
   // the same network as SCL:
   "Output"."5号梯LEDe" := "5号梯数据块"."5号梯2层flag" OR "5号梯数据块"."5号梯6层flag" OR "5号梯数据块"."5号梯8层flag" OR "5号梯数据块"."5号梯10层flag";
END_REGION

REGION Network 7: 5号梯楼层led_f显示
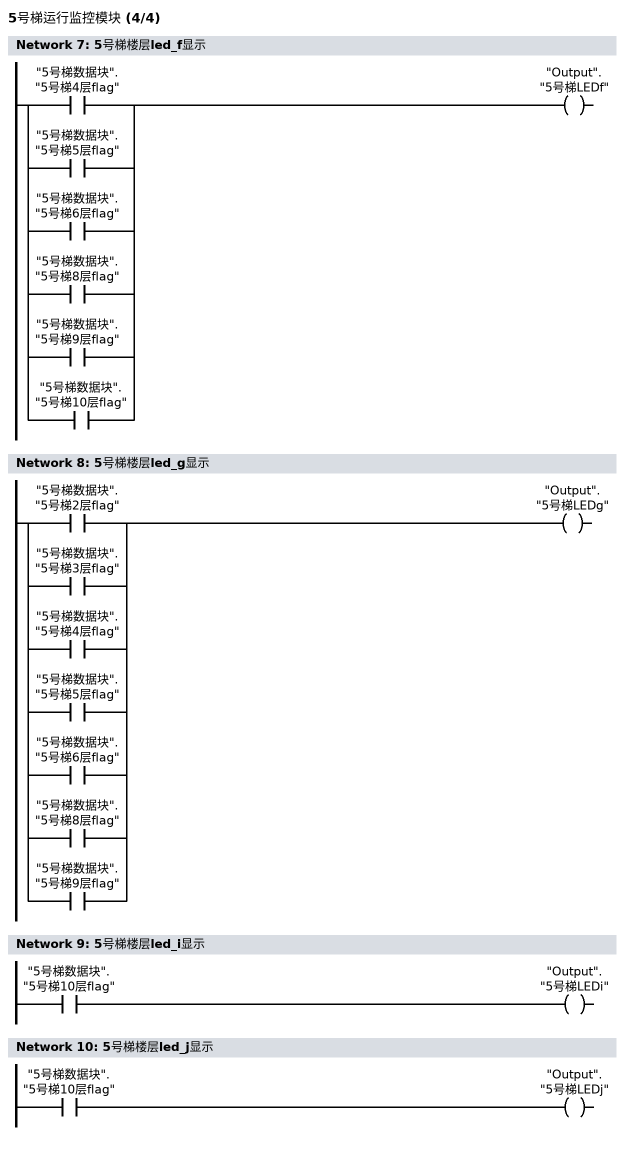
   RUNG wire#powerrail
      Contact( "5号梯数据块"."5号梯4层flag" )
      wire#w1
      Coil( "Output"."5号梯LEDf" )
   END_RUNG
   RUNG wire#powerrail
      Contact( "5号梯数据块"."5号梯5层flag" )
   END_RUNG wire#w1
   RUNG wire#powerrail
      Contact( "5号梯数据块"."5号梯6层flag" )
   END_RUNG wire#w1
   RUNG wire#powerrail
      Contact( "5号梯数据块"."5号梯8层flag" )
   END_RUNG wire#w1
   RUNG wire#powerrail
      Contact( "5号梯数据块"."5号梯9层flag" )
   END_RUNG wire#w1
   RUNG wire#powerrail
      Contact( "5号梯数据块"."5号梯10层flag" )
   END_RUNG wire#w1
   // the same network as SCL:
   "Output"."5号梯LEDf" := "5号梯数据块"."5号梯4层flag" OR "5号梯数据块"."5号梯5层flag" OR "5号梯数据块"."5号梯6层flag" OR "5号梯数据块"."5号梯8层flag" OR "5号梯数据块"."5号梯9层flag" OR "5号梯数据块"."5号梯10层flag";
END_REGION

REGION Network 8: 5号梯楼层led_g显示
   RUNG wire#powerrail
      Contact( "5号梯数据块"."5号梯2层flag" )
      wire#w1
      Coil( "Output"."5号梯LEDg" )
   END_RUNG
   RUNG wire#powerrail
      Contact( "5号梯数据块"."5号梯3层flag" )
   END_RUNG wire#w1
   RUNG wire#powerrail
      Contact( "5号梯数据块"."5号梯4层flag" )
   END_RUNG wire#w1
   RUNG wire#powerrail
      Contact( "5号梯数据块"."5号梯5层flag" )
   END_RUNG wire#w1
   RUNG wire#powerrail
      Contact( "5号梯数据块"."5号梯6层flag" )
   END_RUNG wire#w1
   RUNG wire#powerrail
      Contact( "5号梯数据块"."5号梯8层flag" )
   END_RUNG wire#w1
   RUNG wire#powerrail
      Contact( "5号梯数据块"."5号梯9层flag" )
   END_RUNG wire#w1
   // the same network as SCL:
   "Output"."5号梯LEDg" := "5号梯数据块"."5号梯2层flag" OR "5号梯数据块"."5号梯3层flag" OR "5号梯数据块"."5号梯4层flag" OR "5号梯数据块"."5号梯5层flag" OR "5号梯数据块"."5号梯6层flag" OR "5号梯数据块"."5号梯8层flag" OR "5号梯数据块"."5号梯9层flag";
END_REGION

REGION Network 9: 5号梯楼层led_i显示
   RUNG wire#powerrail
      Contact( "5号梯数据块"."5号梯10层flag" )
      Coil( "Output"."5号梯LEDi" )
   END_RUNG
   // the same network as SCL:
   "Output"."5号梯LEDi" := "5号梯数据块"."5号梯10层flag";
END_REGION

REGION Network 10: 5号梯楼层led_j显示
   RUNG wire#powerrail
      Contact( "5号梯数据块"."5号梯10层flag" )
      Coil( "Output"."5号梯LEDj" )
   END_RUNG
   // the same network as SCL:
   "Output"."5号梯LEDj" := "5号梯数据块"."5号梯10层flag";
END_REGION
END_FUNCTION

FUNCTION "5号梯超重与内选" : Void   // FC24, LAD
{ S7_Optimized_Access := 'TRUE' }
VERSION : 0.1
BEGIN
END_FUNCTION

FUNCTION "5号梯开关门控制" : Void   // FC30, LAD
{ S7_Optimized_Access := 'TRUE' }
VERSION : 0.1
BEGIN
END_FUNCTION

FUNCTION "5号梯楼层计数" : Void   // FC36, LAD
{ S7_Optimized_Access := 'TRUE' }
VERSION : 0.1
BEGIN
END_FUNCTION

FUNCTION "5号梯检修" : Void   // FC53, LAD
{ S7_Optimized_Access := 'TRUE' }
VERSION : 0.1
BEGIN
END_FUNCTION

FUNCTION "5号梯目标楼层与方向判断" : Void   // FC54, LAD
{ S7_Optimized_Access := 'TRUE' }
VERSION : 0.1
BEGIN
END_FUNCTION

FUNCTION "5号梯字节消除与记录" : Void   // FC55, LAD
{ S7_Optimized_Access := 'TRUE' }
VERSION : 0.1
BEGIN
END_FUNCTION

FUNCTION "5号梯启停控制" : Void   // FC62, LAD
{ S7_Optimized_Access := 'TRUE' }
VERSION : 0.1
BEGIN
END_FUNCTION

// folder: 6号梯

FUNCTION "6号梯初始化" : Void   // FC7, LAD
{ S7_Optimized_Access := 'TRUE' }
VERSION : 0.1
   VAR_INPUT
      初始化方向 : Bool;
      初始化楼层 : Byte;
   END_VAR
   VAR_TEMP   // added for the SCL form of the ladder/FBD networks
      _w1 : Bool;
      _w2 : Bool;
      _w3 : Bool;
      _w4 : Bool;
   END_VAR
BEGIN

REGION Network 1: 6号梯传参（方向+初始化楼层）
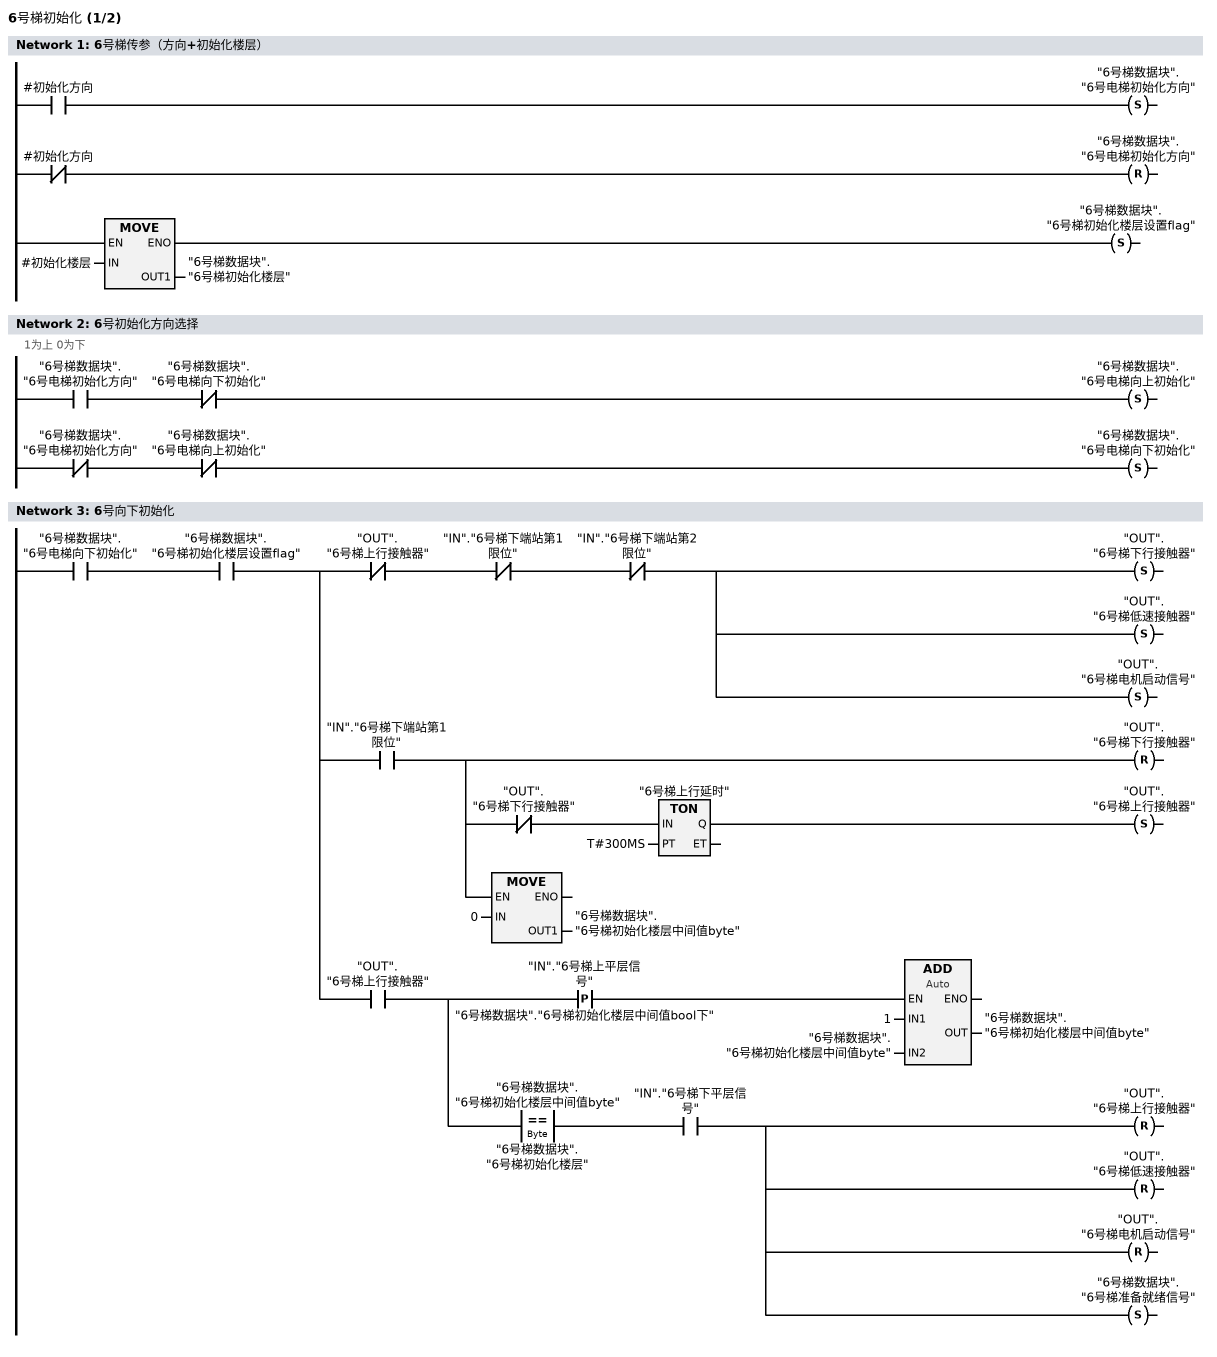
   RUNG wire#powerrail
      Contact( #初始化方向 )
      S_Coil( "6号梯数据块"."6号电梯初始化方向" )
   END_RUNG
   RUNG wire#powerrail
      I_Contact( #初始化方向 )
      R_Coil( "6号梯数据块"."6号电梯初始化方向" )
   END_RUNG
   RUNG wire#powerrail
      Move(in := #初始化楼层, out1 => "6号梯数据块"."6号梯初始化楼层")
      S_Coil( "6号梯数据块"."6号梯初始化楼层设置flag" )
   END_RUNG
   // the same network as SCL:
   IF #初始化方向 THEN "6号梯数据块"."6号电梯初始化方向" := TRUE; END_IF;
   IF NOT #初始化方向 THEN "6号梯数据块"."6号电梯初始化方向" := FALSE; END_IF;
   "6号梯数据块"."6号梯初始化楼层" := #初始化楼层;
   "6号梯数据块"."6号梯初始化楼层设置flag" := TRUE;
END_REGION

REGION Network 2: 6号初始化方向选择
   // 1为上 0为下
   RUNG wire#powerrail
      Contact( "6号梯数据块"."6号电梯初始化方向" )
      I_Contact( "6号梯数据块"."6号电梯向下初始化" )
      S_Coil( "6号梯数据块"."6号电梯向上初始化" )
   END_RUNG
   RUNG wire#powerrail
      I_Contact( "6号梯数据块"."6号电梯初始化方向" )
      I_Contact( "6号梯数据块"."6号电梯向上初始化" )
      S_Coil( "6号梯数据块"."6号电梯向下初始化" )
   END_RUNG
   // the same network as SCL:
   IF "6号梯数据块"."6号电梯初始化方向" AND NOT "6号梯数据块"."6号电梯向下初始化" THEN "6号梯数据块"."6号电梯向上初始化" := TRUE; END_IF;
   IF NOT "6号梯数据块"."6号电梯初始化方向" AND NOT "6号梯数据块"."6号电梯向上初始化" THEN "6号梯数据块"."6号电梯向下初始化" := TRUE; END_IF;
END_REGION

REGION Network 3: 6号向下初始化
   #_w1 := "6号梯数据块"."6号电梯向下初始化" AND "6号梯数据块"."6号梯初始化楼层设置flag";
   IF #_w1 AND NOT "OUT"."6号梯上行接触器" AND NOT "IN"."6号梯下端站第1限位" AND NOT "IN"."6号梯下端站第2限位" THEN
       "OUT"."6号梯下行接触器" := TRUE;
       "OUT"."6号梯低速接触器" := TRUE;
       "OUT"."6号梯电机启动信号" := TRUE;
   END_IF;
   #_w2 := #_w1 AND "IN"."6号梯下端站第1限位";
   IF #_w2 THEN "OUT"."6号梯下行接触器" := FALSE; END_IF;
   "6号梯上行延时".TON(IN := #_w2 AND NOT "OUT"."6号梯下行接触器", PT := T#300MS);
   IF "6号梯上行延时".Q THEN "OUT"."6号梯上行接触器" := TRUE; END_IF;
   IF #_w2 THEN "6号梯数据块"."6号梯初始化楼层中间值byte" := 0; END_IF;
   #_w3 := #_w1 AND "OUT"."6号梯上行接触器";
   #_w4 := #_w3 AND "IN"."6号梯上平层信号" AND NOT "6号梯数据块"."6号梯初始化楼层中间值bool下";   // rising edge of "IN"."6号梯上平层信号"
   "6号梯数据块"."6号梯初始化楼层中间值bool下" := "IN"."6号梯上平层信号";
   IF #_w4 THEN "6号梯数据块"."6号梯初始化楼层中间值byte" := 1 + "6号梯数据块"."6号梯初始化楼层中间值byte"; END_IF;
   IF #_w3 AND ("6号梯数据块"."6号梯初始化楼层中间值byte" = "6号梯数据块"."6号梯初始化楼层") AND "IN"."6号梯下平层信号" THEN
       "OUT"."6号梯上行接触器" := FALSE;
       "OUT"."6号梯低速接触器" := FALSE;
       "OUT"."6号梯电机启动信号" := FALSE;
       "6号梯数据块"."6号梯准备就绪信号" := TRUE;
   END_IF;
END_REGION

REGION Network 4: 6号向上初始化
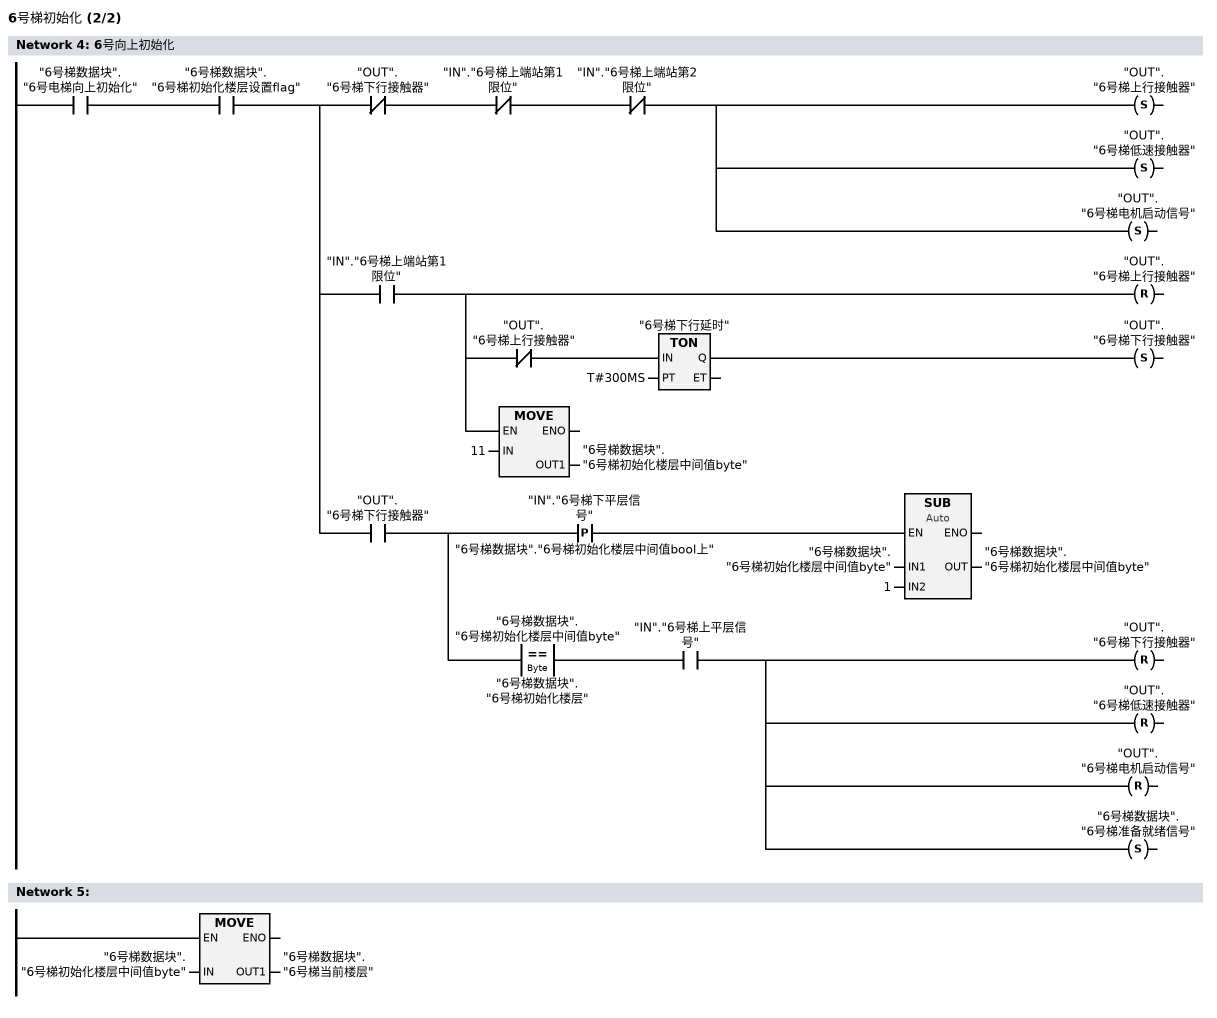
   #_w1 := "6号梯数据块"."6号电梯向上初始化" AND "6号梯数据块"."6号梯初始化楼层设置flag";
   IF #_w1 AND NOT "OUT"."6号梯下行接触器" AND NOT "IN"."6号梯上端站第1限位" AND NOT "IN"."6号梯上端站第2限位" THEN
       "OUT"."6号梯上行接触器" := TRUE;
       "OUT"."6号梯低速接触器" := TRUE;
       "OUT"."6号梯电机启动信号" := TRUE;
   END_IF;
   #_w2 := #_w1 AND "IN"."6号梯上端站第1限位";
   IF #_w2 THEN "OUT"."6号梯上行接触器" := FALSE; END_IF;
   "6号梯下行延时".TON(IN := #_w2 AND NOT "OUT"."6号梯上行接触器", PT := T#300MS);
   IF "6号梯下行延时".Q THEN "OUT"."6号梯下行接触器" := TRUE; END_IF;
   IF #_w2 THEN "6号梯数据块"."6号梯初始化楼层中间值byte" := 11; END_IF;
   #_w3 := #_w1 AND "OUT"."6号梯下行接触器";
   #_w4 := #_w3 AND "IN"."6号梯下平层信号" AND NOT "6号梯数据块"."6号梯初始化楼层中间值bool上";   // rising edge of "IN"."6号梯下平层信号"
   "6号梯数据块"."6号梯初始化楼层中间值bool上" := "IN"."6号梯下平层信号";
   IF #_w4 THEN "6号梯数据块"."6号梯初始化楼层中间值byte" := "6号梯数据块"."6号梯初始化楼层中间值byte" - 1; END_IF;
   IF #_w3 AND ("6号梯数据块"."6号梯初始化楼层中间值byte" = "6号梯数据块"."6号梯初始化楼层") AND "IN"."6号梯上平层信号" THEN
       "OUT"."6号梯下行接触器" := FALSE;
       "OUT"."6号梯低速接触器" := FALSE;
       "OUT"."6号梯电机启动信号" := FALSE;
       "6号梯数据块"."6号梯准备就绪信号" := TRUE;
   END_IF;
END_REGION

REGION Network 5
   RUNG wire#powerrail
      Move(in := "6号梯数据块"."6号梯初始化楼层中间值byte", out1 => "6号梯数据块"."6号梯当前楼层")
   END_RUNG
   // the same network as SCL:
   "6号梯数据块"."6号梯当前楼层" := "6号梯数据块"."6号梯初始化楼层中间值byte";
END_REGION
END_FUNCTION

FUNCTION "6号梯主函数" : Void   // FC12, LAD
{ S7_Optimized_Access := 'TRUE' }
VERSION : 0.1
BEGIN

REGION Network 1
